ABB RAPID module: P80.mod

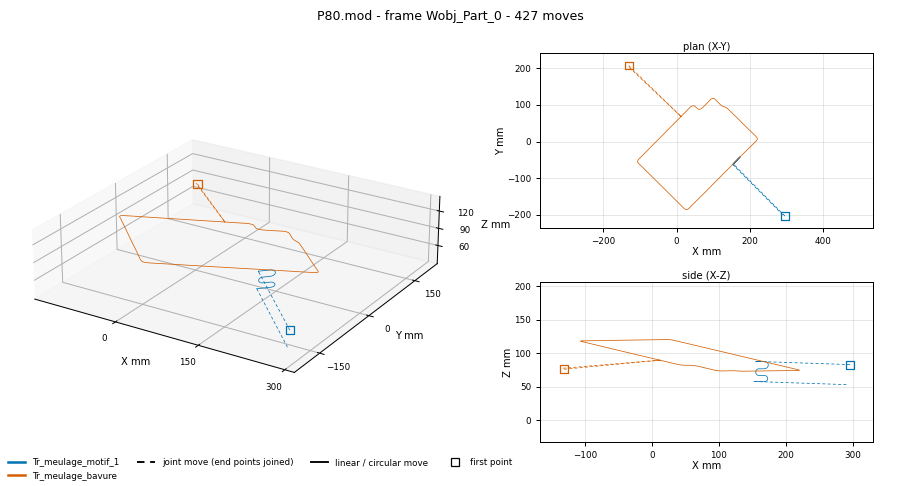
[picture p0: tool path of P80.mod in frame Wobj_Part_0, 427 of 434 moves have a stored position in this frame; points joined in program order, loops and branches not executed]
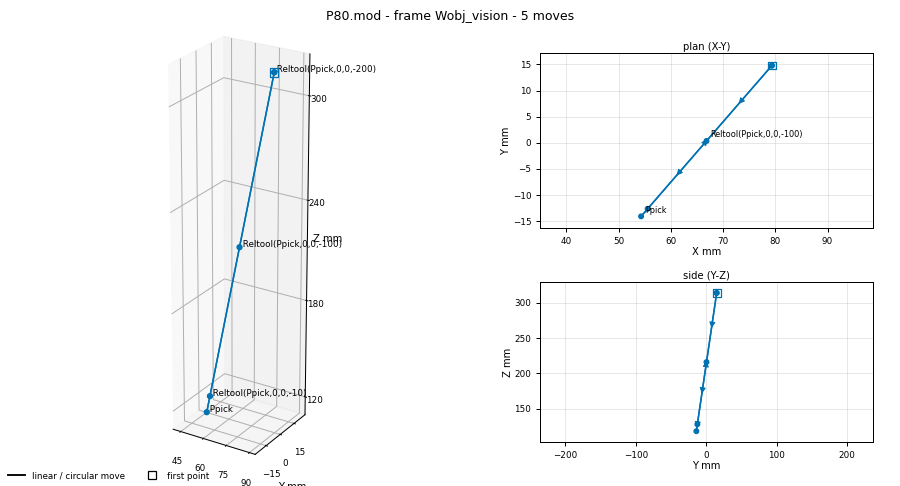
[picture p1: tool path of P80.mod in frame Wobj_vision, 5 of 434 moves have a stored position in this frame; points joined in program order, loops and branches not executed]
MODULE P80
	LOCAL CONST Speeddata vitesse_Tronconnage :=[10, 500, 0, 0];
	LOCAL CONST Robtarget Tr_meulage_motif_1_App1 :=[[295.968307149887,-203.258531598382,82.8714237887279],[0.661524902437711,-0.645987349747704,-0.266117883007714,0.272518659478957],[0,0,0,0],[8.999999E+09,8.999999E+09,8.999999E+09,8.999999E+09,8.999999E+09,8.999999E+09]];
	LOCAL CONST Robtarget Tr_meulage_motif_1_App2 :=[[162.175166138744,-68.4289722830441,87.3864379863114],[0.661524902437711,-0.645987349747704,-0.266117883007714,0.272518659478957],[0,0,0,0],[8.999999E+09,8.999999E+09,8.999999E+09,8.999999E+09,8.999999E+09,8.999999E+09]];
	LOCAL CONST Robtarget Tr_meulage_motif_1_P0 :=[[155.133421875,-61.3326796875,87.6240703125],[0.661524902437711,-0.645987349747704,-0.266117883007714,0.272518659478957],[0,0,0,0],[8.999999E+09,8.999999E+09,8.999999E+09,8.999999E+09,8.999999E+09,8.999999E+09]];
	LOCAL CONST Robtarget Tr_meulage_motif_1_P1 :=[[155.832390625,-60.61752734375,87.6240546875],[0.661524902437711,-0.645987349747704,-0.266117883007714,0.272518659478957],[0,0,0,0],[8.999999E+09,8.999999E+09,8.999999E+09,8.999999E+09,8.999999E+09,8.999999E+09]];
	LOCAL CONST Robtarget Tr_meulage_motif_1_P2 :=[[156.531359375,-59.902375,87.6240390625],[0.661524902437711,-0.645987349747704,-0.266117883007714,0.272518659478957],[0,0,0,0],[8.999999E+09,8.999999E+09,8.999999E+09,8.999999E+09,8.999999E+09,8.999999E+09]];
	LOCAL CONST Robtarget Tr_meulage_motif_1_P3 :=[[157.230328125,-59.18722265625,87.6240234375],[0.661524902437711,-0.645987349747704,-0.266117883007714,0.272518659478957],[0,0,0,0],[8.999999E+09,8.999999E+09,8.999999E+09,8.999999E+09,8.999999E+09,8.999999E+09]];
	LOCAL CONST Robtarget Tr_meulage_motif_1_P4 :=[[157.929296875,-58.47207421875,87.6240078125],[0.661524902437711,-0.645987349747704,-0.266117883007714,0.272518659478957],[0,0,0,0],[8.999999E+09,8.999999E+09,8.999999E+09,8.999999E+09,8.999999E+09,8.999999E+09]];
	LOCAL CONST Robtarget Tr_meulage_motif_1_P5 :=[[158.628265625,-57.756921875,87.6239921875],[0.661524902437711,-0.645987349747704,-0.266117883007714,0.272518659478957],[0,0,0,0],[8.999999E+09,8.999999E+09,8.999999E+09,8.999999E+09,8.999999E+09,8.999999E+09]];
	LOCAL CONST Robtarget Tr_meulage_motif_1_P6 :=[[159.327234375,-57.04176953125,87.6239765625],[0.661524902437711,-0.645987349747704,-0.266117883007714,0.272518659478957],[0,0,0,0],[8.999999E+09,8.999999E+09,8.999999E+09,8.999999E+09,8.999999E+09,8.999999E+09]];
	LOCAL CONST Robtarget Tr_meulage_motif_1_P7 :=[[160.026203125,-56.3266171875,87.6239609375],[0.661524902437711,-0.645987349747704,-0.266117883007714,0.272518659478957],[0,0,0,0],[8.999999E+09,8.999999E+09,8.999999E+09,8.999999E+09,8.999999E+09,8.999999E+09]];
	LOCAL CONST Robtarget Tr_meulage_motif_1_P8 :=[[160.725171875,-55.61146484375,87.6239453125],[0.661524902437711,-0.645987349747704,-0.266117883007714,0.272518659478957],[0,0,0,0],[8.999999E+09,8.999999E+09,8.999999E+09,8.999999E+09,8.999999E+09,8.999999E+09]];
	LOCAL CONST Robtarget Tr_meulage_motif_1_P9 :=[[161.424140625,-54.8963125,87.6239296875],[0.661524902437711,-0.645987349747704,-0.266117883007714,0.272518659478957],[0,0,0,0],[8.999999E+09,8.999999E+09,8.999999E+09,8.999999E+09,8.999999E+09,8.999999E+09]];
	LOCAL CONST Robtarget Tr_meulage_motif_1_P10 :=[[162.123109375,-54.1811640625,87.6239140625],[0.661524902437711,-0.645987349747704,-0.266117883007714,0.272518659478957],[0,0,0,0],[8.999999E+09,8.999999E+09,8.999999E+09,8.999999E+09,8.999999E+09,8.999999E+09]];
	LOCAL CONST Robtarget Tr_meulage_motif_1_P11 :=[[162.822078125,-53.46601171875,87.623890625],[0.661524902437711,-0.645987349747704,-0.266117883007714,0.272518659478957],[0,0,0,0],[8.999999E+09,8.999999E+09,8.999999E+09,8.999999E+09,8.999999E+09,8.999999E+09]];
	LOCAL CONST Robtarget Tr_meulage_motif_1_P12 :=[[163.521046875,-52.750859375,87.623875],[0.661524902437711,-0.645987349747704,-0.266117883007714,0.272518659478957],[0,0,0,0],[8.999999E+09,8.999999E+09,8.999999E+09,8.999999E+09,8.999999E+09,8.999999E+09]];
	LOCAL CONST Robtarget Tr_meulage_motif_1_P13 :=[[164.220015625,-52.03570703125,87.623859375],[0.661524902437711,-0.645987349747704,-0.266117883007714,0.272518659478957],[0,0,0,0],[8.999999E+09,8.999999E+09,8.999999E+09,8.999999E+09,8.999999E+09,8.999999E+09]];
	LOCAL CONST Robtarget Tr_meulage_motif_1_P14 :=[[164.918984375,-51.3205546875,87.62384375],[0.661524902437711,-0.645987349747704,-0.266117883007714,0.272518659478957],[0,0,0,0],[8.999999E+09,8.999999E+09,8.999999E+09,8.999999E+09,8.999999E+09,8.999999E+09]];
	LOCAL CONST Robtarget Tr_meulage_motif_1_P15 :=[[165.617953125,-50.60540625,87.623828125],[0.661524902437711,-0.645987349747704,-0.266117883007714,0.272518659478957],[0,0,0,0],[8.999999E+09,8.999999E+09,8.999999E+09,8.999999E+09,8.999999E+09,8.999999E+09]];
	LOCAL CONST Robtarget Tr_meulage_motif_1_P16 :=[[166.316921875,-49.89025390625,87.6238125],[0.661524902437711,-0.645987349747704,-0.266117883007714,0.272518659478957],[0,0,0,0],[8.999999E+09,8.999999E+09,8.999999E+09,8.999999E+09,8.999999E+09,8.999999E+09]];
	LOCAL CONST Robtarget Tr_meulage_motif_1_P17 :=[[167.015890625,-49.1751015625,87.623796875],[0.661524902437711,-0.645987349747704,-0.266117883007714,0.272518659478957],[0,0,0,0],[8.999999E+09,8.999999E+09,8.999999E+09,8.999999E+09,8.999999E+09,8.999999E+09]];
	LOCAL CONST Robtarget Tr_meulage_motif_1_P18 :=[[167.714859375,-48.45994921875,87.62378125],[0.661524902437711,-0.645987349747704,-0.266117883007714,0.272518659478957],[0,0,0,0],[8.999999E+09,8.999999E+09,8.999999E+09,8.999999E+09,8.999999E+09,8.999999E+09]];
	LOCAL CONST Robtarget Tr_meulage_motif_1_P19 :=[[168.413828125,-47.744796875,87.623765625],[0.661524902437711,-0.645987349747704,-0.266117883007714,0.272518659478957],[0,0,0,0],[8.999999E+09,8.999999E+09,8.999999E+09,8.999999E+09,8.999999E+09,8.999999E+09]];
	LOCAL CONST Robtarget Tr_meulage_motif_1_P20 :=[[169.1128125,-47.0296484375,87.62375],[0.661524902437711,-0.645987349747704,-0.266117883007714,0.272518659478957],[0,0,0,0],[8.999999E+09,8.999999E+09,8.999999E+09,8.999999E+09,8.999999E+09,8.999999E+09]];
	LOCAL CONST Robtarget Tr_meulage_motif_1_P21 :=[[169.80340625,-46.31671484375,87.5132265625],[0.661524902437711,-0.645987349747704,-0.266117883007714,0.272518659478957],[0,0,0,0],[8.999999E+09,8.999999E+09,8.999999E+09,8.999999E+09,8.999999E+09,8.999999E+09]];
	LOCAL CONST Robtarget Tr_meulage_motif_1_P22 :=[[170.458921875,-45.63391015625,87.3021953125],[0.661524902437711,-0.645987349747704,-0.266117883007714,0.272518659478957],[0,0,0,0],[8.999999E+09,8.999999E+09,8.999999E+09,8.999999E+09,8.999999E+09,8.999999E+09]];
	LOCAL CONST Robtarget Tr_meulage_motif_1_P23 :=[[171.047140625,-45.01647265625,87.0305546875],[0.661524902437711,-0.645987349747704,-0.266117883007714,0.272518659478957],[0,0,0,0],[8.999999E+09,8.999999E+09,8.999999E+09,8.999999E+09,8.999999E+09,8.999999E+09]];
	LOCAL CONST Robtarget Tr_meulage_motif_1_P24 :=[[171.563421875,-44.47242578125,86.754828125],[0.661524902437711,-0.645987349747704,-0.266117883007714,0.272518659478957],[0,0,0,0],[8.999999E+09,8.999999E+09,8.999999E+09,8.999999E+09,8.999999E+09,8.999999E+09]];
	LOCAL CONST Robtarget Tr_meulage_motif_1_P25 :=[[172.315359375,-43.66773828125,86.1391796875],[0.661524902437711,-0.645987349747704,-0.266117883007714,0.272518659478957],[0,0,0,0],[8.999999E+09,8.999999E+09,8.999999E+09,8.999999E+09,8.999999E+09,8.999999E+09]];
	LOCAL CONST Robtarget Tr_meulage_motif_1_P26 :=[[173.006703125,-42.91176953125,85.2921953125],[0.661524902437711,-0.645987349747704,-0.266117883007714,0.272518659478957],[0,0,0,0],[8.999999E+09,8.999999E+09,8.999999E+09,8.999999E+09,8.999999E+09,8.999999E+09]];
	LOCAL CONST Robtarget Tr_meulage_motif_1_P27 :=[[173.5698125,-42.27688671875,84.269125],[0.661524902437711,-0.645987349747704,-0.266117883007714,0.272518659478957],[0,0,0,0],[8.999999E+09,8.999999E+09,8.999999E+09,8.999999E+09,8.999999E+09,8.999999E+09]];
	LOCAL CONST Robtarget Tr_meulage_motif_1_P28 :=[[173.879015625,-41.896515625,83.153828125],[0.661524902437711,-0.645987349747704,-0.266117883007714,0.272518659478957],[0,0,0,0],[8.999999E+09,8.999999E+09,8.999999E+09,8.999999E+09,8.999999E+09,8.999999E+09]];
	LOCAL CONST Robtarget Tr_meulage_motif_1_P29 :=[[173.87796875,-41.85766796875,82.458421875],[0.661524902437711,-0.645987349747704,-0.266117883007714,0.272518659478957],[0,0,0,0],[8.999999E+09,8.999999E+09,8.999999E+09,8.999999E+09,8.999999E+09,8.999999E+09]];
	LOCAL CONST Robtarget Tr_meulage_motif_1_P30 :=[[173.859,-41.83914453125,81.797703125],[0.661524902437711,-0.645987349747704,-0.266117883007714,0.272518659478957],[0,0,0,0],[8.999999E+09,8.999999E+09,8.999999E+09,8.999999E+09,8.999999E+09,8.999999E+09]];
	LOCAL CONST Robtarget Tr_meulage_motif_1_P31 :=[[173.801671875,-41.85987109375,81.137140625],[0.661524902437711,-0.645987349747704,-0.266117883007714,0.272518659478957],[0,0,0,0],[8.999999E+09,8.999999E+09,8.999999E+09,8.999999E+09,8.999999E+09,8.999999E+09]];
	LOCAL CONST Robtarget Tr_meulage_motif_1_P32 :=[[173.42184375,-42.1853125,80.03628125],[0.661524902437711,-0.645987349747704,-0.266117883007714,0.272518659478957],[0,0,0,0],[8.999999E+09,8.999999E+09,8.999999E+09,8.999999E+09,8.999999E+09,8.999999E+09]];
	LOCAL CONST Robtarget Tr_meulage_motif_1_P33 :=[[172.79421875,-42.76973046875,79.030484375],[0.661524902437711,-0.645987349747704,-0.266117883007714,0.272518659478957],[0,0,0,0],[8.999999E+09,8.999999E+09,8.999999E+09,8.999999E+09,8.999999E+09,8.999999E+09]];
	LOCAL CONST Robtarget Tr_meulage_motif_1_P34 :=[[172.055109375,-43.47840625,78.2022890625],[0.661524902437711,-0.645987349747704,-0.266117883007714,0.272518659478957],[0,0,0,0],[8.999999E+09,8.999999E+09,8.999999E+09,8.999999E+09,8.999999E+09,8.999999E+09]];
	LOCAL CONST Robtarget Tr_meulage_motif_1_P35 :=[[171.5635,-43.9586953125,77.8068671875],[0.661524902437711,-0.645987349747704,-0.266117883007714,0.272518659478957],[0,0,0,0],[8.999999E+09,8.999999E+09,8.999999E+09,8.999999E+09,8.999999E+09,8.999999E+09]];
	LOCAL CONST Robtarget Tr_meulage_motif_1_P36 :=[[170.74,-44.773296875,77.31975],[0.661524902437711,-0.645987349747704,-0.266117883007714,0.272518659478957],[0,0,0,0],[8.999999E+09,8.999999E+09,8.999999E+09,8.999999E+09,8.999999E+09,8.999999E+09]];
	LOCAL CONST Robtarget Tr_meulage_motif_1_P37 :=[[170.14178125,-45.3702265625,77.0558828125],[0.661524902437711,-0.645987349747704,-0.266117883007714,0.272518659478957],[0,0,0,0],[8.999999E+09,8.999999E+09,8.999999E+09,8.999999E+09,8.999999E+09,8.999999E+09]];
	LOCAL CONST Robtarget Tr_meulage_motif_1_P38 :=[[169.48446875,-46.03101953125,76.85159375],[0.661524902437711,-0.645987349747704,-0.266117883007714,0.272518659478957],[0,0,0,0],[8.999999E+09,8.999999E+09,8.999999E+09,8.999999E+09,8.999999E+09,8.999999E+09]];
	LOCAL CONST Robtarget Tr_meulage_motif_1_P39 :=[[168.795265625,-46.72994140625,76.7431015625],[0.661524902437711,-0.645987349747704,-0.266117883007714,0.272518659478957],[0,0,0,0],[8.999999E+09,8.999999E+09,8.999999E+09,8.999999E+09,8.999999E+09,8.999999E+09]];
	LOCAL CONST Robtarget Tr_meulage_motif_1_P40 :=[[168.098328125,-47.43667578125,76.632609375],[0.661524902437711,-0.645987349747704,-0.266117883007714,0.272518659478957],[0,0,0,0],[8.999999E+09,8.999999E+09,8.999999E+09,8.999999E+09,8.999999E+09,8.999999E+09]];
	LOCAL CONST Robtarget Tr_meulage_motif_1_P41 :=[[167.399359375,-48.151828125,76.632625],[0.661524902437711,-0.645987349747704,-0.266117883007714,0.272518659478957],[0,0,0,0],[8.999999E+09,8.999999E+09,8.999999E+09,8.999999E+09,8.999999E+09,8.999999E+09]];
	LOCAL CONST Robtarget Tr_meulage_motif_1_P42 :=[[166.700390625,-48.86698046875,76.632640625],[0.661524902437711,-0.645987349747704,-0.266117883007714,0.272518659478957],[0,0,0,0],[8.999999E+09,8.999999E+09,8.999999E+09,8.999999E+09,8.999999E+09,8.999999E+09]];
	LOCAL CONST Robtarget Tr_meulage_motif_1_P43 :=[[166.001421875,-49.5821328125,76.63265625],[0.661524902437711,-0.645987349747704,-0.266117883007714,0.272518659478957],[0,0,0,0],[8.999999E+09,8.999999E+09,8.999999E+09,8.999999E+09,8.999999E+09,8.999999E+09]];
	LOCAL CONST Robtarget Tr_meulage_motif_1_P44 :=[[165.302453125,-50.29728515625,76.632671875],[0.661524902437711,-0.645987349747704,-0.266117883007714,0.272518659478957],[0,0,0,0],[8.999999E+09,8.999999E+09,8.999999E+09,8.999999E+09,8.999999E+09,8.999999E+09]];
	LOCAL CONST Robtarget Tr_meulage_motif_1_P45 :=[[164.603484375,-51.01243359375,76.6326875],[0.661524902437711,-0.645987349747704,-0.266117883007714,0.272518659478957],[0,0,0,0],[8.999999E+09,8.999999E+09,8.999999E+09,8.999999E+09,8.999999E+09,8.999999E+09]];
	LOCAL CONST Robtarget Tr_meulage_motif_1_P46 :=[[163.904515625,-51.7275859375,76.632703125],[0.661524902437711,-0.645987349747704,-0.266117883007714,0.272518659478957],[0,0,0,0],[8.999999E+09,8.999999E+09,8.999999E+09,8.999999E+09,8.999999E+09,8.999999E+09]];
	LOCAL CONST Robtarget Tr_meulage_motif_1_P47 :=[[163.205546875,-52.44273828125,76.63271875],[0.661524902437711,-0.645987349747704,-0.266117883007714,0.272518659478957],[0,0,0,0],[8.999999E+09,8.999999E+09,8.999999E+09,8.999999E+09,8.999999E+09,8.999999E+09]];
	LOCAL CONST Robtarget Tr_meulage_motif_1_P48 :=[[162.506578125,-53.157890625,76.632734375],[0.661524902437711,-0.645987349747704,-0.266117883007714,0.272518659478957],[0,0,0,0],[8.999999E+09,8.999999E+09,8.999999E+09,8.999999E+09,8.999999E+09,8.999999E+09]];
	LOCAL CONST Robtarget Tr_meulage_motif_1_P49 :=[[161.807609375,-53.87304296875,76.6327578125],[0.661524902437711,-0.645987349747704,-0.266117883007714,0.272518659478957],[0,0,0,0],[8.999999E+09,8.999999E+09,8.999999E+09,8.999999E+09,8.999999E+09,8.999999E+09]];
	LOCAL CONST Robtarget Tr_meulage_motif_1_P50 :=[[161.108640625,-54.58819140625,76.6327734375],[0.661524902437711,-0.645987349747704,-0.266117883007714,0.272518659478957],[0,0,0,0],[8.999999E+09,8.999999E+09,8.999999E+09,8.999999E+09,8.999999E+09,8.999999E+09]];
	LOCAL CONST Robtarget Tr_meulage_motif_1_P51 :=[[160.409671875,-55.30334375,76.6327890625],[0.661524902437711,-0.645987349747704,-0.266117883007714,0.272518659478957],[0,0,0,0],[8.999999E+09,8.999999E+09,8.999999E+09,8.999999E+09,8.999999E+09,8.999999E+09]];
	LOCAL CONST Robtarget Tr_meulage_motif_1_P52 :=[[159.710703125,-56.01849609375,76.6328046875],[0.661524902437711,-0.645987349747704,-0.266117883007714,0.272518659478957],[0,0,0,0],[8.999999E+09,8.999999E+09,8.999999E+09,8.999999E+09,8.999999E+09,8.999999E+09]];
	LOCAL CONST Robtarget Tr_meulage_motif_1_P53 :=[[159.01375,-56.72523046875,76.5223125],[0.661524902437711,-0.645987349747704,-0.266117883007714,0.272518659478957],[0,0,0,0],[8.999999E+09,8.999999E+09,8.999999E+09,8.999999E+09,8.999999E+09,8.999999E+09]];
	LOCAL CONST Robtarget Tr_meulage_motif_1_P54 :=[[158.346125,-57.39620703125,76.3113125],[0.661524902437711,-0.645987349747704,-0.266117883007714,0.272518659478957],[0,0,0,0],[8.999999E+09,8.999999E+09,8.999999E+09,8.999999E+09,8.999999E+09,8.999999E+09]];
	LOCAL CONST Robtarget Tr_meulage_motif_1_P55 :=[[157.742296875,-57.9984140625,76.0396953125],[0.661524902437711,-0.645987349747704,-0.266117883007714,0.272518659478957],[0,0,0,0],[8.999999E+09,8.999999E+09,8.999999E+09,8.999999E+09,8.999999E+09,8.999999E+09]];
	LOCAL CONST Robtarget Tr_meulage_motif_1_P56 :=[[157.236265625,-58.4987265625,75.735796875],[0.661524902437711,-0.645987349747704,-0.266117883007714,0.272518659478957],[0,0,0,0],[8.999999E+09,8.999999E+09,8.999999E+09,8.999999E+09,8.999999E+09,8.999999E+09]];
	LOCAL CONST Robtarget Tr_meulage_motif_1_P57 :=[[156.494203125,-59.21996875,75.0738125],[0.661524902437711,-0.645987349747704,-0.266117883007714,0.272518659478957],[0,0,0,0],[8.999999E+09,8.999999E+09,8.999999E+09,8.999999E+09,8.999999E+09,8.999999E+09]];
	LOCAL CONST Robtarget Tr_meulage_motif_1_P58 :=[[155.83790625,-59.8397265625,74.1726171875],[0.661524902437711,-0.645987349747704,-0.266117883007714,0.272518659478957],[0,0,0,0],[8.999999E+09,8.999999E+09,8.999999E+09,8.999999E+09,8.999999E+09,8.999999E+09]];
	LOCAL CONST Robtarget Tr_meulage_motif_1_P59 :=[[155.43396875,-60.19301171875,73.1274375],[0.661524902437711,-0.645987349747704,-0.266117883007714,0.272518659478957],[0,0,0,0],[8.999999E+09,8.999999E+09,8.999999E+09,8.999999E+09,8.999999E+09,8.999999E+09]];
	LOCAL CONST Robtarget Tr_meulage_motif_1_P60 :=[[155.2849375,-60.30573828125,72.43478125],[0.661524902437711,-0.645987349747704,-0.266117883007714,0.272518659478957],[0,0,0,0],[8.999999E+09,8.999999E+09,8.999999E+09,8.999999E+09,8.999999E+09,8.999999E+09]];
	LOCAL CONST Robtarget Tr_meulage_motif_1_P61 :=[[155.21821875,-60.329828125,71.6653984375],[0.661524902437711,-0.645987349747704,-0.266117883007714,0.272518659478957],[0,0,0,0],[8.999999E+09,8.999999E+09,8.999999E+09,8.999999E+09,8.999999E+09,8.999999E+09]];
	LOCAL CONST Robtarget Tr_meulage_motif_1_P62 :=[[155.242921875,-60.26039453125,70.896140625],[0.661524902437711,-0.645987349747704,-0.266117883007714,0.272518659478957],[0,0,0,0],[8.999999E+09,8.999999E+09,8.999999E+09,8.999999E+09,8.999999E+09,8.999999E+09]];
	LOCAL CONST Robtarget Tr_meulage_motif_1_P63 :=[[155.504421875,-59.92927734375,69.7887734375],[0.661524902437711,-0.645987349747704,-0.266117883007714,0.272518659478957],[0,0,0,0],[8.999999E+09,8.999999E+09,8.999999E+09,8.999999E+09,8.999999E+09,8.999999E+09]];
	LOCAL CONST Robtarget Tr_meulage_motif_1_P64 :=[[155.77721875,-59.61657421875,69.2035546875],[0.661524902437711,-0.645987349747704,-0.266117883007714,0.272518659478957],[0,0,0,0],[8.999999E+09,8.999999E+09,8.999999E+09,8.999999E+09,8.999999E+09,8.999999E+09]];
	LOCAL CONST Robtarget Tr_meulage_motif_1_P65 :=[[156.37184375,-58.957296875,68.317125],[0.661524902437711,-0.645987349747704,-0.266117883007714,0.272518659478957],[0,0,0,0],[8.999999E+09,8.999999E+09,8.999999E+09,8.999999E+09,8.999999E+09,8.999999E+09]];
	LOCAL CONST Robtarget Tr_meulage_motif_1_P66 :=[[156.76934375,-58.5268359375,67.903140625],[0.661524902437711,-0.645987349747704,-0.266117883007714,0.272518659478957],[0,0,0,0],[8.999999E+09,8.999999E+09,8.999999E+09,8.999999E+09,8.999999E+09,8.999999E+09]];
	LOCAL CONST Robtarget Tr_meulage_motif_1_P67 :=[[157.535109375,-57.712125,67.3594609375],[0.661524902437711,-0.645987349747704,-0.266117883007714,0.272518659478957],[0,0,0,0],[8.999999E+09,8.999999E+09,8.999999E+09,8.999999E+09,8.999999E+09,8.999999E+09]];
	LOCAL CONST Robtarget Tr_meulage_motif_1_P68 :=[[158.103703125,-57.113421875,67.0641875],[0.661524902437711,-0.645987349747704,-0.266117883007714,0.272518659478957],[0,0,0,0],[8.999999E+09,8.999999E+09,8.999999E+09,8.999999E+09,8.999999E+09,8.999999E+09]];
	LOCAL CONST Robtarget Tr_meulage_motif_1_P69 :=[[158.74928125,-56.441171875,66.8598671875],[0.661524902437711,-0.645987349747704,-0.266117883007714,0.272518659478957],[0,0,0,0],[8.999999E+09,8.999999E+09,8.999999E+09,8.999999E+09,8.999999E+09,8.999999E+09]];
	LOCAL CONST Robtarget Tr_meulage_motif_1_P70 :=[[159.43225,-55.7361640625,66.75134375],[0.661524902437711,-0.645987349747704,-0.266117883007714,0.272518659478957],[0,0,0,0],[8.999999E+09,8.999999E+09,8.999999E+09,8.999999E+09,8.999999E+09,8.999999E+09]];
	LOCAL CONST Robtarget Tr_meulage_motif_1_P71 :=[[160.12284375,-55.023234375,66.640828125],[0.661524902437711,-0.645987349747704,-0.266117883007714,0.272518659478957],[0,0,0,0],[8.999999E+09,8.999999E+09,8.999999E+09,8.999999E+09,8.999999E+09,8.999999E+09]];
	LOCAL CONST Robtarget Tr_meulage_motif_1_P72 :=[[160.8218125,-54.30808203125,66.6408125],[0.661524902437711,-0.645987349747704,-0.266117883007714,0.272518659478957],[0,0,0,0],[8.999999E+09,8.999999E+09,8.999999E+09,8.999999E+09,8.999999E+09,8.999999E+09]];
	LOCAL CONST Robtarget Tr_meulage_motif_1_P73 :=[[161.52078125,-53.59293359375,66.640796875],[0.661524902437711,-0.645987349747704,-0.266117883007714,0.272518659478957],[0,0,0,0],[8.999999E+09,8.999999E+09,8.999999E+09,8.999999E+09,8.999999E+09,8.999999E+09]];
	LOCAL CONST Robtarget Tr_meulage_motif_1_P74 :=[[162.21975,-52.87778125,66.64078125],[0.661524902437711,-0.645987349747704,-0.266117883007714,0.272518659478957],[0,0,0,0],[8.999999E+09,8.999999E+09,8.999999E+09,8.999999E+09,8.999999E+09,8.999999E+09]];
	LOCAL CONST Robtarget Tr_meulage_motif_1_P75 :=[[162.91871875,-52.16262890625,66.640765625],[0.661524902437711,-0.645987349747704,-0.266117883007714,0.272518659478957],[0,0,0,0],[8.999999E+09,8.999999E+09,8.999999E+09,8.999999E+09,8.999999E+09,8.999999E+09]];
	LOCAL CONST Robtarget Tr_meulage_motif_1_P76 :=[[163.6176875,-51.4474765625,66.6407421875],[0.661524902437711,-0.645987349747704,-0.266117883007714,0.272518659478957],[0,0,0,0],[8.999999E+09,8.999999E+09,8.999999E+09,8.999999E+09,8.999999E+09,8.999999E+09]];
	LOCAL CONST Robtarget Tr_meulage_motif_1_P77 :=[[164.31665625,-50.73232421875,66.6407265625],[0.661524902437711,-0.645987349747704,-0.266117883007714,0.272518659478957],[0,0,0,0],[8.999999E+09,8.999999E+09,8.999999E+09,8.999999E+09,8.999999E+09,8.999999E+09]];
	LOCAL CONST Robtarget Tr_meulage_motif_1_P78 :=[[165.015625,-50.01717578125,66.6407109375],[0.661524902437711,-0.645987349747704,-0.266117883007714,0.272518659478957],[0,0,0,0],[8.999999E+09,8.999999E+09,8.999999E+09,8.999999E+09,8.999999E+09,8.999999E+09]];
	LOCAL CONST Robtarget Tr_meulage_motif_1_P79 :=[[165.71459375,-49.3020234375,66.6406953125],[0.661524902437711,-0.645987349747704,-0.266117883007714,0.272518659478957],[0,0,0,0],[8.999999E+09,8.999999E+09,8.999999E+09,8.999999E+09,8.999999E+09,8.999999E+09]];
	LOCAL CONST Robtarget Tr_meulage_motif_1_P80 :=[[166.4135625,-48.58687109375,66.6406796875],[0.661524902437711,-0.645987349747704,-0.266117883007714,0.272518659478957],[0,0,0,0],[8.999999E+09,8.999999E+09,8.999999E+09,8.999999E+09,8.999999E+09,8.999999E+09]];
	LOCAL CONST Robtarget Tr_meulage_motif_1_P81 :=[[167.11253125,-47.87171875,66.6406640625],[0.661524902437711,-0.645987349747704,-0.266117883007714,0.272518659478957],[0,0,0,0],[8.999999E+09,8.999999E+09,8.999999E+09,8.999999E+09,8.999999E+09,8.999999E+09]];
	LOCAL CONST Robtarget Tr_meulage_motif_1_P82 :=[[167.8115,-47.15656640625,66.6406484375],[0.661524902437711,-0.645987349747704,-0.266117883007714,0.272518659478957],[0,0,0,0],[8.999999E+09,8.999999E+09,8.999999E+09,8.999999E+09,8.999999E+09,8.999999E+09]];
	LOCAL CONST Robtarget Tr_meulage_motif_1_P83 :=[[168.51046875,-46.4414140625,66.6406328125],[0.661524902437711,-0.645987349747704,-0.266117883007714,0.272518659478957],[0,0,0,0],[8.999999E+09,8.999999E+09,8.999999E+09,8.999999E+09,8.999999E+09,8.999999E+09]];
	LOCAL CONST Robtarget Tr_meulage_motif_1_P84 :=[[169.201078125,-45.728484375,66.530109375],[0.661524902437711,-0.645987349747704,-0.266117883007714,0.272518659478957],[0,0,0,0],[8.999999E+09,8.999999E+09,8.999999E+09,8.999999E+09,8.999999E+09,8.999999E+09]];
	LOCAL CONST Robtarget Tr_meulage_motif_1_P85 :=[[169.85659375,-45.0456796875,66.319078125],[0.661524902437711,-0.645987349747704,-0.266117883007714,0.272518659478957],[0,0,0,0],[8.999999E+09,8.999999E+09,8.999999E+09,8.999999E+09,8.999999E+09,8.999999E+09]];
	LOCAL CONST Robtarget Tr_meulage_motif_1_P86 :=[[170.4448125,-44.4282421875,66.0474453125],[0.661524902437711,-0.645987349747704,-0.266117883007714,0.272518659478957],[0,0,0,0],[8.999999E+09,8.999999E+09,8.999999E+09,8.999999E+09,8.999999E+09,8.999999E+09]];
	LOCAL CONST Robtarget Tr_meulage_motif_1_P87 :=[[170.96109375,-43.88419140625,65.7717109375],[0.661524902437711,-0.645987349747704,-0.266117883007714,0.272518659478957],[0,0,0,0],[8.999999E+09,8.999999E+09,8.999999E+09,8.999999E+09,8.999999E+09,8.999999E+09]];
	LOCAL CONST Robtarget Tr_meulage_motif_1_P88 :=[[171.71303125,-43.0795078125,65.15606640625],[0.661524902437711,-0.645987349747704,-0.266117883007714,0.272518659478957],[0,0,0,0],[8.999999E+09,8.999999E+09,8.999999E+09,8.999999E+09,8.999999E+09,8.999999E+09]];
	LOCAL CONST Robtarget Tr_meulage_motif_1_P89 :=[[172.404375,-42.3235390625,64.30907421875],[0.661524902437711,-0.645987349747704,-0.266117883007714,0.272518659478957],[0,0,0,0],[8.999999E+09,8.999999E+09,8.999999E+09,8.999999E+09,8.999999E+09,8.999999E+09]];
	LOCAL CONST Robtarget Tr_meulage_motif_1_P90 :=[[172.89975,-41.7556015625,63.24498046875],[0.661524902437711,-0.645987349747704,-0.266117883007714,0.272518659478957],[0,0,0,0],[8.999999E+09,8.999999E+09,8.999999E+09,8.999999E+09,8.999999E+09,8.999999E+09]];
	LOCAL CONST Robtarget Tr_meulage_motif_1_P91 :=[[173.087890625,-41.50144140625,62.17071484375],[0.661524902437711,-0.645987349747704,-0.266117883007714,0.272518659478957],[0,0,0,0],[8.999999E+09,8.999999E+09,8.999999E+09,8.999999E+09,8.999999E+09,8.999999E+09]];
	LOCAL CONST Robtarget Tr_meulage_motif_1_P92 :=[[173.030015625,-41.5273515625,61.59058984375],[0.661524902437711,-0.645987349747704,-0.266117883007714,0.272518659478957],[0,0,0,0],[8.999999E+09,8.999999E+09,8.999999E+09,8.999999E+09,8.999999E+09,8.999999E+09]];
	LOCAL CONST Robtarget Tr_meulage_motif_1_P93 :=[[173.021046875,-41.5125625,61.17301953125],[0.661524902437711,-0.645987349747704,-0.266117883007714,0.272518659478957],[0,0,0,0],[8.999999E+09,8.999999E+09,8.999999E+09,8.999999E+09,8.999999E+09,8.999999E+09]];
	LOCAL CONST Robtarget Tr_meulage_motif_1_P94 :=[[172.740109375,-41.74440625,60.2044921875],[0.661524902437711,-0.645987349747704,-0.266117883007714,0.272518659478957],[0,0,0,0],[8.999999E+09,8.999999E+09,8.999999E+09,8.999999E+09,8.999999E+09,8.999999E+09]];
	LOCAL CONST Robtarget Tr_meulage_motif_1_P95 :=[[172.13928125,-42.30651171875,59.2875859375],[0.661524902437711,-0.645987349747704,-0.266117883007714,0.272518659478957],[0,0,0,0],[8.999999E+09,8.999999E+09,8.999999E+09,8.999999E+09,8.999999E+09,8.999999E+09]];
	LOCAL CONST Robtarget Tr_meulage_motif_1_P96 :=[[171.699265625,-42.73244921875,58.865],[0.661524902437711,-0.645987349747704,-0.266117883007714,0.272518659478957],[0,0,0,0],[8.999999E+09,8.999999E+09,8.999999E+09,8.999999E+09,8.999999E+09,8.999999E+09]];
	LOCAL CONST Robtarget Tr_meulage_motif_1_P97 :=[[170.894,-43.5259375,58.3350078125],[0.661524902437711,-0.645987349747704,-0.266117883007714,0.272518659478957],[0,0,0,0],[8.999999E+09,8.999999E+09,8.999999E+09,8.999999E+09,8.999999E+09,8.999999E+09]];
	LOCAL CONST Robtarget Tr_meulage_motif_1_P98 :=[[170.29578125,-44.12286328125,58.071140625],[0.661524902437711,-0.645987349747704,-0.266117883007714,0.272518659478957],[0,0,0,0],[8.999999E+09,8.999999E+09,8.999999E+09,8.999999E+09,8.999999E+09,8.999999E+09]];
	LOCAL CONST Robtarget Tr_meulage_motif_1_P99 :=[[169.63846875,-44.78365625,57.86684765625],[0.661524902437711,-0.645987349747704,-0.266117883007714,0.272518659478957],[0,0,0,0],[8.999999E+09,8.999999E+09,8.999999E+09,8.999999E+09,8.999999E+09,8.999999E+09]];
	LOCAL CONST Robtarget Tr_meulage_motif_1_P100 :=[[168.94928125,-45.48258203125,57.758359375],[0.661524902437711,-0.645987349747704,-0.266117883007714,0.272518659478957],[0,0,0,0],[8.999999E+09,8.999999E+09,8.999999E+09,8.999999E+09,8.999999E+09,8.999999E+09]];
	LOCAL CONST Robtarget Tr_meulage_motif_1_P101 :=[[168.252328125,-46.18931640625,57.64787109375],[0.661524902437711,-0.645987349747704,-0.266117883007714,0.272518659478957],[0,0,0,0],[8.999999E+09,8.999999E+09,8.999999E+09,8.999999E+09,8.999999E+09,8.999999E+09]];
	LOCAL CONST Robtarget Tr_meulage_motif_1_P102 :=[[167.553359375,-46.90446875,57.64788671875],[0.661524902437711,-0.645987349747704,-0.266117883007714,0.272518659478957],[0,0,0,0],[8.999999E+09,8.999999E+09,8.999999E+09,8.999999E+09,8.999999E+09,8.999999E+09]];
	LOCAL CONST Robtarget Tr_meulage_motif_1_P103 :=[[166.854390625,-47.61962109375,57.64790234375],[0.661524902437711,-0.645987349747704,-0.266117883007714,0.272518659478957],[0,0,0,0],[8.999999E+09,8.999999E+09,8.999999E+09,8.999999E+09,8.999999E+09,8.999999E+09]];
	LOCAL CONST Robtarget Tr_meulage_motif_1_P104 :=[[166.155421875,-48.3347734375,57.64791796875],[0.661524902437711,-0.645987349747704,-0.266117883007714,0.272518659478957],[0,0,0,0],[8.999999E+09,8.999999E+09,8.999999E+09,8.999999E+09,8.999999E+09,8.999999E+09]];
	LOCAL CONST Robtarget Tr_meulage_motif_1_P105 :=[[165.456453125,-49.049921875,57.64793359375],[0.661524902437711,-0.645987349747704,-0.266117883007714,0.272518659478957],[0,0,0,0],[8.999999E+09,8.999999E+09,8.999999E+09,8.999999E+09,8.999999E+09,8.999999E+09]];
	LOCAL CONST Robtarget Tr_meulage_motif_1_P106 :=[[164.757484375,-49.76507421875,57.64794921875],[0.661524902437711,-0.645987349747704,-0.266117883007714,0.272518659478957],[0,0,0,0],[8.999999E+09,8.999999E+09,8.999999E+09,8.999999E+09,8.999999E+09,8.999999E+09]];
	LOCAL CONST Robtarget Tr_meulage_motif_1_P107 :=[[164.058515625,-50.4802265625,57.64796484375],[0.661524902437711,-0.645987349747704,-0.266117883007714,0.272518659478957],[0,0,0,0],[8.999999E+09,8.999999E+09,8.999999E+09,8.999999E+09,8.999999E+09,8.999999E+09]];
	LOCAL CONST Robtarget Tr_meulage_motif_1_P108 :=[[163.359546875,-51.19537890625,57.64798046875],[0.661524902437711,-0.645987349747704,-0.266117883007714,0.272518659478957],[0,0,0,0],[8.999999E+09,8.999999E+09,8.999999E+09,8.999999E+09,8.999999E+09,8.999999E+09]];
	LOCAL CONST Robtarget Tr_meulage_motif_1_P109 :=[[162.660578125,-51.91053125,57.64799609375],[0.661524902437711,-0.645987349747704,-0.266117883007714,0.272518659478957],[0,0,0,0],[8.999999E+09,8.999999E+09,8.999999E+09,8.999999E+09,8.999999E+09,8.999999E+09]];
	LOCAL CONST Robtarget Tr_meulage_motif_1_P110 :=[[161.961609375,-52.6256796875,57.64801171875],[0.661524902437711,-0.645987349747704,-0.266117883007714,0.272518659478957],[0,0,0,0],[8.999999E+09,8.999999E+09,8.999999E+09,8.999999E+09,8.999999E+09,8.999999E+09]];
	LOCAL CONST Robtarget Tr_meulage_motif_1_P111 :=[[161.262640625,-53.34083203125,57.64803125],[0.661524902437711,-0.645987349747704,-0.266117883007714,0.272518659478957],[0,0,0,0],[8.999999E+09,8.999999E+09,8.999999E+09,8.999999E+09,8.999999E+09,8.999999E+09]];
	LOCAL CONST Robtarget Tr_meulage_motif_1_P112 :=[[160.563671875,-54.055984375,57.648046875],[0.661524902437711,-0.645987349747704,-0.266117883007714,0.272518659478957],[0,0,0,0],[8.999999E+09,8.999999E+09,8.999999E+09,8.999999E+09,8.999999E+09,8.999999E+09]];
	LOCAL CONST Robtarget Tr_meulage_motif_1_P113 :=[[159.864703125,-54.77113671875,57.6480625],[0.661524902437711,-0.645987349747704,-0.266117883007714,0.272518659478957],[0,0,0,0],[8.999999E+09,8.999999E+09,8.999999E+09,8.999999E+09,8.999999E+09,8.999999E+09]];
	LOCAL CONST Robtarget Tr_meulage_motif_1_P114 :=[[159.165734375,-55.4862890625,57.648078125],[0.661524902437711,-0.645987349747704,-0.266117883007714,0.272518659478957],[0,0,0,0],[8.999999E+09,8.999999E+09,8.999999E+09,8.999999E+09,8.999999E+09,8.999999E+09]];
	LOCAL CONST Robtarget Tr_meulage_motif_1_P115 :=[[158.466765625,-56.2014375,57.64809375],[0.661524902437711,-0.645987349747704,-0.266117883007714,0.272518659478957],[0,0,0,0],[8.999999E+09,8.999999E+09,8.999999E+09,8.999999E+09,8.999999E+09,8.999999E+09]];
	LOCAL CONST Robtarget Tr_meulage_motif_1_P116 :=[[157.767796875,-56.91658984375,57.648109375],[0.661524902437711,-0.645987349747704,-0.266117883007714,0.272518659478957],[0,0,0,0],[8.999999E+09,8.999999E+09,8.999999E+09,8.999999E+09,8.999999E+09,8.999999E+09]];
	LOCAL CONST Robtarget Tr_meulage_motif_1_P117 :=[[157.068828125,-57.6317421875,57.648125],[0.661524902437711,-0.645987349747704,-0.266117883007714,0.272518659478957],[0,0,0,0],[8.999999E+09,8.999999E+09,8.999999E+09,8.999999E+09,8.999999E+09,8.999999E+09]];
	LOCAL CONST Robtarget Tr_meulage_motif_1_P118 :=[[156.369859375,-58.34689453125,57.648140625],[0.661524902437711,-0.645987349747704,-0.266117883007714,0.272518659478957],[0,0,0,0],[8.999999E+09,8.999999E+09,8.999999E+09,8.999999E+09,8.999999E+09,8.999999E+09]];
	LOCAL CONST Robtarget Tr_meulage_motif_1_P119 :=[[155.670890625,-59.062046875,57.64815625],[0.661524902437711,-0.645987349747704,-0.266117883007714,0.272518659478957],[0,0,0,0],[8.999999E+09,8.999999E+09,8.999999E+09,8.999999E+09,8.999999E+09,8.999999E+09]];
	LOCAL CONST Robtarget Tr_meulage_motif_1_P120 :=[[154.971921875,-59.7771953125,57.648171875],[0.661524902437711,-0.645987349747704,-0.266117883007714,0.272518659478957],[0,0,0,0],[8.999999E+09,8.999999E+09,8.999999E+09,8.999999E+09,8.999999E+09,8.999999E+09]];
	LOCAL CONST Robtarget Tr_meulage_motif_1_P121 :=[[154.272953125,-60.49234765625,57.6481875],[0.661524902437711,-0.645987349747704,-0.266117883007714,0.272518659478957],[0,0,0,0],[8.999999E+09,8.999999E+09,8.999999E+09,8.999999E+09,8.999999E+09,8.999999E+09]];
	LOCAL CONST Robtarget Tr_meulage_motif_1_P122 :=[[153.573984375,-61.2075,57.64820703125],[0.661524902437711,-0.645987349747704,-0.266117883007714,0.272518659478957],[0,0,0,0],[8.999999E+09,8.999999E+09,8.999999E+09,8.999999E+09,8.999999E+09,8.999999E+09]];
	LOCAL CONST Robtarget Tr_meulage_motif_1_P123 :=[[152.875015625,-61.92265234375,57.64822265625],[0.661524902437711,-0.645987349747704,-0.266117883007714,0.272518659478957],[0,0,0,0],[8.999999E+09,8.999999E+09,8.999999E+09,8.999999E+09,8.999999E+09,8.999999E+09]];
	LOCAL CONST Robtarget Tr_meulage_motif_1_degg1 :=[[159.916759888744,-69.0189449392941,57.4105903300614],[0.661524902437711,-0.645987349747704,-0.266117883007714,0.272518659478957],[0,0,0,0],[8.999999E+09,8.999999E+09,8.999999E+09,8.999999E+09,8.999999E+09,8.999999E+09]];
	LOCAL CONST Robtarget Tr_meulage_motif_1_degg2 :=[[293.709900899887,-203.848504254632,52.8955761324779],[0.661524902437711,-0.645987349747704,-0.266117883007714,0.272518659478957],[0,0,0,0],[8.999999E+09,8.999999E+09,8.999999E+09,8.999999E+09,8.999999E+09,8.999999E+09]];
	LOCAL CONST Robtarget Tr_meulage_bavure_App1 :=[[-130.802481498914,207.516367832347,75.9567690677868],[0.284428212423492,-0.265826681388466,0.628943133613018,-0.672954160489858],[0,0,0,0],[8.999999E+09,8.999999E+09,8.999999E+09,8.999999E+09,8.999999E+09,8.999999E+09]];
	LOCAL CONST Robtarget Tr_meulage_bavure_App2 :=[[5.1532886203668,75.4126773759924,88.7881189221393],[0.284428212423492,-0.265826681388466,0.628943133613018,-0.672954160489858],[0,0,0,0],[8.999999E+09,8.999999E+09,8.999999E+09,8.999999E+09,8.999999E+09,8.999999E+09]];
	LOCAL CONST Robtarget Tr_meulage_bavure_P0 :=[[12.30885546875,68.4598515625,89.463453125],[0.284428212423492,-0.265826681388466,0.628943133613018,-0.672954160489858],[0,0,0,0],[8.999999E+09,8.999999E+09,8.999999E+09,8.999999E+09,8.999999E+09,8.999999E+09]];
	LOCAL CONST Robtarget Tr_meulage_bavure_P1 :=[[12.0715,68.21390625,89.5204921875],[0.284373042901133,-0.26576929181495,0.628958710011008,-0.672985584615762],[0,0,0,0],[8.999999E+09,8.999999E+09,8.999999E+09,8.999999E+09,8.999999E+09,8.999999E+09]];
	LOCAL CONST Robtarget Tr_meulage_bavure_P2 :=[[8.9287109375,65.15151953125,90.2510546875],[0.284222180764744,-0.265608224533555,0.62899684472372,-0.673077255854831],[0,0,0,0],[8.999999E+09,8.999999E+09,8.999999E+09,8.999999E+09,8.999999E+09,8.999999E+09]];
	LOCAL CONST Robtarget Tr_meulage_bavure_P3 :=[[4.699265625,60.7726875,91.266953125],[0.284001346399506,-0.26537480227308,0.629055039986907,-0.673208144802825],[0,0,0,0],[8.999999E+09,8.999999E+09,8.999999E+09,8.999999E+09,8.999999E+09,8.999999E+09]];
	LOCAL CONST Robtarget Tr_meulage_bavure_P4 :=[[3.99077392578125,60.0665703125,91.4336484375],[0.283733376273213,-0.265091369093486,0.629125242398549,-0.673367185566472],[0,0,0,0],[8.999999E+09,8.999999E+09,8.999999E+09,8.999999E+09,8.999999E+09,8.999999E+09]];
	LOCAL CONST Robtarget Tr_meulage_bavure_P5 :=[[3.88059838867188,59.94528125,91.46103125],[0.28347686519291,-0.264814256821455,0.629186003163786,-0.673527467670979],[0,0,0,0],[8.999999E+09,8.999999E+09,8.999999E+09,8.999999E+09,8.999999E+09,8.999999E+09]];
	LOCAL CONST Robtarget Tr_meulage_bavure_P6 :=[[3.76301000976563,59.827015625,91.488828125],[0.283331719588849,-0.264646166761516,0.629208160231015,-0.673633902199083],[0,0,0,0],[8.999999E+09,8.999999E+09,8.999999E+09,8.999999E+09,8.999999E+09,8.999999E+09]];
	LOCAL CONST Robtarget Tr_meulage_bavure_P7 :=[[3.63213793945313,59.70169921875,91.51896875],[0.283479615359356,-0.264761899820276,0.629125995315525,-0.673602943949564],[0,0,0,0],[8.999999E+09,8.999999E+09,8.999999E+09,8.999999E+09,8.999999E+09,8.999999E+09]];
	LOCAL CONST Robtarget Tr_meulage_bavure_P8 :=[[3.41819189453125,59.48340234375,91.569953125],[0.284213845397937,-0.265440258548562,0.628829065072101,-0.673303769591659],[0,0,0,0],[8.999999E+09,8.999999E+09,8.999999E+09,8.999999E+09,8.999999E+09,8.999999E+09]];
	LOCAL CONST Robtarget Tr_meulage_bavure_P9 :=[[-0.958820983886719,55.14005859375,92.5973671875],[0.285807861531897,-0.266942308684276,0.628212680896572,-0.67261021229358],[0,0,0,0],[8.999999E+09,8.999999E+09,8.999999E+09,8.999999E+09,8.999999E+09,8.999999E+09]];
	LOCAL CONST Robtarget Tr_meulage_bavure_P10 :=[[-6.55028466796875,49.414171875,93.9323984375],[0.288322350056615,-0.269327080784598,0.627247398799099,-0.67148629674301],[0,0,0,0],[8.999999E+09,8.999999E+09,8.999999E+09,8.999999E+09,8.999999E+09,8.999999E+09]];
	LOCAL CONST Robtarget Tr_meulage_bavure_P11 :=[[-8.520876953125,47.44456640625,94.3967578125],[0.29141978931461,-0.272289487305219,0.62606789240698,-0.67005368113008],[0,0,0,0],[8.999999E+09,8.999999E+09,8.999999E+09,8.999999E+09,8.999999E+09,8.999999E+09]];
	LOCAL CONST Robtarget Tr_meulage_bavure_P12 :=[[-9.8624462890625,46.0195546875,94.723578125],[0.294369215143396,-0.275146476809444,0.624964034618918,-0.668626305875005],[0,0,0,0],[8.999999E+09,8.999999E+09,8.999999E+09,8.999999E+09,8.999999E+09,8.999999E+09]];
	LOCAL CONST Robtarget Tr_meulage_bavure_P13 :=[[-11.689984375,44.16079296875,95.1583125],[0.296268636909546,-0.277054979800622,0.624311920199916,-0.667607713592144],[0,0,0,0],[8.999999E+09,8.999999E+09,8.999999E+09,8.999999E+09,8.999999E+09,8.999999E+09]];
	LOCAL CONST Robtarget Tr_meulage_bavure_P14 :=[[-11.7441982421875,44.07610546875,95.1749609375],[0.29642432777975,-0.277366079829103,0.624411730781714,-0.667316016683807],[0,0,0,0],[8.999999E+09,8.999999E+09,8.999999E+09,8.999999E+09,8.999999E+09,8.999999E+09]];
	LOCAL CONST Robtarget Tr_meulage_bavure_P15 :=[[-14.0992275390625,41.6959140625,95.7332578125],[0.294687475657803,-0.275932746223752,0.625323368688705,-0.667825647773175],[0,0,0,0],[8.999999E+09,8.999999E+09,8.999999E+09,8.999999E+09,8.999999E+09,8.999999E+09]];
	LOCAL CONST Robtarget Tr_meulage_bavure_P16 :=[[-14.4200859375,41.392875,95.806625],[0.291523045570414,-0.273182110372919,0.626838877391853,-0.668923665498292],[0,0,0,0],[8.999999E+09,8.999999E+09,8.999999E+09,8.999999E+09,8.999999E+09,8.999999E+09]];
	LOCAL CONST Robtarget Tr_meulage_bavure_P17 :=[[-15.989626953125,39.8081171875,96.1785078125],[0.28777160038532,-0.269893857490973,0.628595285599939,-0.670233376236849],[0,0,0,0],[8.999999E+09,8.999999E+09,8.999999E+09,8.999999E+09,8.999999E+09,8.999999E+09]];
	LOCAL CONST Robtarget Tr_meulage_bavure_P18 :=[[-20.5275,35.3738203125,97.234953125],[0.284306583970974,-0.266879921516261,0.630230152784219,-0.671382773329649],[0,0,0,0],[8.999999E+09,8.999999E+09,8.999999E+09,8.999999E+09,8.999999E+09,8.999999E+09]];
	LOCAL CONST Robtarget Tr_meulage_bavure_P19 :=[[-21.675865234375,34.22190234375,97.5060859375],[0.281736631260211,-0.264703803449232,0.631499517747391,-0.672134455395994],[0,0,0,0],[8.999999E+09,8.999999E+09,8.999999E+09,8.999999E+09,8.999999E+09,8.999999E+09]];
	LOCAL CONST Robtarget Tr_meulage_bavure_P20 :=[[-25.820263671875,30.174119140625,98.470671875],[0.280280494877072,-0.263565603698652,0.632319207039449,-0.672419836967524],[0,0,0,0],[8.999999E+09,8.999999E+09,8.999999E+09,8.999999E+09,8.999999E+09,8.999999E+09]];
	LOCAL CONST Robtarget Tr_meulage_bavure_P21 :=[[-29.943333984375,25.966017578125,99.4533203125],[0.279831511777758,-0.263365067852669,0.632734307370033,-0.672294922134697],[0,0,0,0],[8.999999E+09,8.999999E+09,8.999999E+09,8.999999E+09,8.999999E+09,8.999999E+09]];
	LOCAL CONST Robtarget Tr_meulage_bavure_P22 :=[[-30.65425390625,25.273341796875,99.6185703125],[0.280098455209423,-0.263823147198514,0.632852238379101,-0.671893032238115],[0,0,0,0],[8.999999E+09,8.999999E+09,8.999999E+09,8.999999E+09,8.999999E+09,8.999999E+09]];
	LOCAL CONST Robtarget Tr_meulage_bavure_P23 :=[[-31.59001953125,24.25621875,99.8494765625],[0.280755004027766,-0.264628999192664,0.632794717727717,-0.671356064779009],[0,0,0,0],[8.999999E+09,8.999999E+09,8.999999E+09,8.999999E+09,8.999999E+09,8.999999E+09]];
	LOCAL CONST Robtarget Tr_meulage_bavure_P24 :=[[-33.03751171875,22.785212890625,100.1936484375],[0.281494324913843,-0.265490782989762,0.632678385129633,-0.670815660355766],[0,0,0,0],[8.999999E+09,8.999999E+09,8.999999E+09,8.999999E+09,8.999999E+09,8.999999E+09]];
	LOCAL CONST Robtarget Tr_meulage_bavure_P25 :=[[-35.58303125,20.01735546875,100.8218984375],[0.282069674309091,-0.266177353782537,0.632602905091275,-0.670372940711787],[0,0,0,0],[8.999999E+09,8.999999E+09,8.999999E+09,8.999999E+09,8.999999E+09,8.999999E+09]];
	LOCAL CONST Robtarget Tr_meulage_bavure_P26 :=[[-35.98186328125,19.596505859375,100.918703125],[0.28234267845556,-0.266560840783109,0.632627454835272,-0.670082407970981],[0,0,0,0],[8.999999E+09,8.999999E+09,8.999999E+09,8.999999E+09,8.999999E+09,8.999999E+09]];
	LOCAL CONST Robtarget Tr_meulage_bavure_P27 :=[[-35.99944140625,19.584302734375,100.9221640625],[0.282265557944378,-0.26659776528805,0.632774037575629,-0.669961792725529],[0,0,0,0],[8.999999E+09,8.999999E+09,8.999999E+09,8.999999E+09,8.999999E+09,8.999999E+09]];
	LOCAL CONST Robtarget Tr_meulage_bavure_P28 :=[[-36.72640234375,18.841884765625,101.0954765625],[0.281868959392986,-0.266325730096396,0.633040201901723,-0.669985520735756],[0,0,0,0],[8.999999E+09,8.999999E+09,8.999999E+09,8.999999E+09,8.999999E+09,8.999999E+09]];
	LOCAL CONST Robtarget Tr_meulage_bavure_P29 :=[[-40.45190234375,15.164779296875,101.967453125],[0.281268755948015,-0.265862992961441,0.633389182694683,-0.670091709504306],[0,0,0,0],[8.999999E+09,8.999999E+09,8.999999E+09,8.999999E+09,8.999999E+09,8.999999E+09]];
	LOCAL CONST Robtarget Tr_meulage_bavure_P30 :=[[-46.5366875,9.034759765625,103.4074296875],[0.280629008001166,-0.265374589995516,0.633766366094151,-0.670196896487001],[0,0,0,0],[8.999999E+09,8.999999E+09,8.999999E+09,8.999999E+09,8.999999E+09,8.999999E+09]];
	LOCAL CONST Robtarget Tr_meulage_bavure_P31 :=[[-47.9009765625,7.66512158203125,103.7296875],[0.280126846706262,-0.265044675438766,0.634119448740969,-0.670203547069407],[0,0,0,0],[8.999999E+09,8.999999E+09,8.999999E+09,8.999999E+09,8.999999E+09,8.999999E+09]];
	LOCAL CONST Robtarget Tr_meulage_bavure_P32 :=[[-49.00028515625,6.58895849609375,103.985859375],[0.279912301482713,-0.26502575630409,0.634400388606441,-0.670034774403607],[0,0,0,0],[8.999999E+09,8.999999E+09,8.999999E+09,8.999999E+09,8.999999E+09,8.999999E+09]];
	LOCAL CONST Robtarget Tr_meulage_bavure_P33 :=[[-56.24496875,-0.754955444335938,105.70609375],[0.280039190285508,-0.265387076054559,0.634606547332694,-0.669643399019154],[0,0,0,0],[8.999999E+09,8.999999E+09,8.999999E+09,8.999999E+09,8.999999E+09,8.999999E+09]];
	LOCAL CONST Robtarget Tr_meulage_bavure_P34 :=[[-56.44252734375,-0.940341125488281,105.751109375],[0.280436694311137,-0.266076323772035,0.634779618441978,-0.669039226370516],[0,0,0,0],[8.999999E+09,8.999999E+09,8.999999E+09,8.999999E+09,8.999999E+09,8.999999E+09]];
	LOCAL CONST Robtarget Tr_meulage_bavure_P35 :=[[-61.49255859375,-6.014634765625,106.9445234375],[0.28089986869357,-0.266914266221368,0.635014623407983,-0.668287712226899],[0,0,0,0],[8.999999E+09,8.999999E+09,8.999999E+09,8.999999E+09,8.999999E+09,8.999999E+09]];
	LOCAL CONST Robtarget Tr_meulage_bavure_P36 :=[[-62.0686875,-6.60664013671875,107.08234375],[0.281135980929385,-0.267639959443632,0.635445326692624,-0.66748831384556],[0,0,0,0],[8.999999E+09,8.999999E+09,8.999999E+09,8.999999E+09,8.999999E+09,8.999999E+09]];
	LOCAL CONST Robtarget Tr_meulage_bavure_P37 :=[[-62.15234765625,-6.68784228515625,107.10175],[0.280872409861467,-0.268002066607424,0.636191141596299,-0.666743138717722],[0,0,0,0],[8.999999E+09,8.999999E+09,8.999999E+09,8.999999E+09,8.999999E+09,8.999999E+09]];
	LOCAL CONST Robtarget Tr_meulage_bavure_P38 :=[[-62.4766171875,-7.02322021484375,107.17959375],[0.279952648313818,-0.267860150951519,0.637328446406798,-0.666100522169895],[0,0,0,0],[8.999999E+09,8.999999E+09,8.999999E+09,8.999999E+09,8.999999E+09,8.999999E+09]];
	LOCAL CONST Robtarget Tr_meulage_bavure_P39 :=[[-63.384140625,-7.966861328125,107.39809375],[0.278409568963992,-0.267250326223849,0.638854365642366,-0.665530220607765],[0,0,0,0],[8.999999E+09,8.999999E+09,8.999999E+09,8.999999E+09,8.999999E+09,8.999999E+09]];
	LOCAL CONST Robtarget Tr_meulage_bavure_P40 :=[[-76.2720078125,-21.096939453125,110.4666328125],[0.27647060340918,-0.2663891523062,0.64068105745596,-0.6649275205624],[0,0,0,0],[8.999999E+09,8.999999E+09,8.999999E+09,8.999999E+09,8.999999E+09,8.999999E+09]];
	LOCAL CONST Robtarget Tr_meulage_bavure_P41 :=[[-80.59846875,-25.452609375,111.490125],[0.274546255000979,-0.26567165495655,0.642647017176692,-0.664114249908467],[0,0,0,0],[8.999999E+09,8.999999E+09,8.999999E+09,8.999999E+09,8.999999E+09,8.999999E+09]];
	LOCAL CONST Robtarget Tr_meulage_bavure_P42 :=[[-83.3634140625,-28.0718984375,112.1233359375],[0.273144744796606,-0.265588810037895,0.644546334529159,-0.662883515421584],[0,0,0,0],[8.999999E+09,8.999999E+09,8.999999E+09,8.999999E+09,8.999999E+09,8.999999E+09]];
	LOCAL CONST Robtarget Tr_meulage_bavure_P43 :=[[-86.130109375,-30.768453125,112.7665546875],[0.272817776514206,-0.266688663135384,0.646156350621466,-0.661006496431355],[0,0,0,0],[8.999999E+09,8.999999E+09,8.999999E+09,8.999999E+09,8.999999E+09,8.999999E+09]];
	LOCAL CONST Robtarget Tr_meulage_bavure_P44 :=[[-86.8596484375,-31.48644140625,112.9370390625],[0.27428351230221,-0.269688662603679,0.647164415709515,-0.658190549295236],[0,0,0,0],[8.999999E+09,8.999999E+09,8.999999E+09,8.999999E+09,8.999999E+09,8.999999E+09]];
	LOCAL CONST Robtarget Tr_meulage_bavure_P45 :=[[-88.19725,-32.81711328125,113.2514453125],[0.278407617210333,-0.275468154571829,0.647155596433672,-0.65406125745272],[0,0,0,0],[8.999999E+09,8.999999E+09,8.999999E+09,8.999999E+09,8.999999E+09,8.999999E+09]];
	LOCAL CONST Robtarget Tr_meulage_bavure_P46 :=[[-91.98925,-36.439203125,114.12365625],[0.286353616651651,-0.285230997494903,0.645506962357269,-0.648047564494207],[0,0,0,0],[8.999999E+09,8.999999E+09,8.999999E+09,8.999999E+09,8.999999E+09,8.999999E+09]];
	LOCAL CONST Robtarget Tr_meulage_bavure_P47 :=[[-95.3056484375,-39.89283203125,114.922796875],[0.299650668113211,-0.300587306240852,0.641254795041416,-0.639256627859709],[0,0,0,0],[8.999999E+09,8.999999E+09,8.999999E+09,8.999999E+09,8.999999E+09,8.999999E+09]];
	LOCAL CONST Robtarget Tr_meulage_bavure_P48 :=[[-100.4908984375,-45.2673359375,116.169046875],[0.320051028593992,-0.323416808300398,0.632955064228461,-0.626367938094101],[0,0,0,0],[8.999999E+09,8.999999E+09,8.999999E+09,8.999999E+09,8.999999E+09,8.999999E+09]];
	LOCAL CONST Robtarget Tr_meulage_bavure_P49 :=[[-103.1467109375,-47.98748046875,116.8032109375],[0.349083003066893,-0.355430902110319,0.618610109095904,-0.607561901141931],[0,0,0,0],[8.999999E+09,8.999999E+09,8.999999E+09,8.999999E+09,8.999999E+09,8.999999E+09]];
	LOCAL CONST Robtarget Tr_meulage_bavure_P50 :=[[-104.90665625,-50.2904921875,117.2870546875],[0.387058512056147,-0.397136430194387,0.595929379738561,-0.580806799565702],[0,0,0,0],[8.999999E+09,8.999999E+09,8.999999E+09,8.999999E+09,8.999999E+09,8.999999E+09]];
	LOCAL CONST Robtarget Tr_meulage_bavure_P51 :=[[-105.5893203125,-51.99621875,117.57796875],[0.43184428563275,-0.44652973010744,0.563316451820981,-0.544790132256759],[0,0,0,0],[8.999999E+09,8.999999E+09,8.999999E+09,8.999999E+09,8.999999E+09,8.999999E+09]];
	LOCAL CONST Robtarget Tr_meulage_bavure_P52 :=[[-106.2798515625,-54.09439453125,117.9196015625],[0.478392482158397,-0.498481197686526,0.52160530549503,-0.500584691982057],[0,0,0,0],[8.999999E+09,8.999999E+09,8.999999E+09,8.999999E+09,8.999999E+09,8.999999E+09]];
	LOCAL CONST Robtarget Tr_meulage_bavure_P53 :=[[-106.24278125,-54.8323671875,118.0093515625],[0.520658622167301,-0.546637683470221,0.474882966311317,-0.452314061776242],[0,0,0,0],[8.999999E+09,8.999999E+09,8.999999E+09,8.999999E+09,8.999999E+09,8.999999E+09]];
	LOCAL CONST Robtarget Tr_meulage_bavure_P54 :=[[-105.2187578125,-57.02176953125,118.1763203125],[0.554709056689723,-0.586678986818574,0.42871377759736,-0.405351854257668],[0,0,0,0],[8.999999E+09,8.999999E+09,8.999999E+09,8.999999E+09,8.999999E+09,8.999999E+09]];
	LOCAL CONST Robtarget Tr_meulage_bavure_P55 :=[[-104.978359375,-57.656765625,118.2308984375],[0.579801101572751,-0.617550876730381,0.387462675636133,-0.363777778669137],[0,0,0,0],[8.999999E+09,8.999999E+09,8.999999E+09,8.999999E+09,8.999999E+09,8.999999E+09]];
	LOCAL CONST Robtarget Tr_meulage_bavure_P56 :=[[-104.8231328125,-57.89610546875,118.2444453125],[0.597111227807004,-0.640236934194449,0.353422853377421,-0.329616650718174],[0,0,0,0],[8.999999E+09,8.999999E+09,8.999999E+09,8.999999E+09,8.999999E+09,8.999999E+09]];
	LOCAL CONST Robtarget Tr_meulage_bavure_P57 :=[[-103.4312578125,-59.53333203125,118.3012890625],[0.608331665190778,-0.656340290957888,0.327298218171311,-0.303357683227926],[0,0,0,0],[8.999999E+09,8.999999E+09,8.999999E+09,8.999999E+09,8.999999E+09,8.999999E+09]];
	LOCAL CONST Robtarget Tr_meulage_bavure_P58 :=[[-102.9890546875,-59.9969296875,118.31215625],[0.615011742863901,-0.667368044766304,0.308835564102726,-0.284606822317489],[0,0,0,0],[8.999999E+09,8.999999E+09,8.999999E+09,8.999999E+09,8.999999E+09,8.999999E+09]];
	LOCAL CONST Robtarget Tr_meulage_bavure_P59 :=[[-100.397296875,-62.29012109375,118.3220078125],[0.61845408506239,-0.674611894552726,0.297063956793492,-0.272334981175422],[0,0,0,0],[8.999999E+09,8.999999E+09,8.999999E+09,8.999999E+09,8.999999E+09,8.999999E+09]];
	LOCAL CONST Robtarget Tr_meulage_bavure_P60 :=[[-95.87471875,-66.59021875,118.377125],[0.619715785437852,-0.67915851952747,0.29053891952191,-0.265109763825179],[0,0,0,0],[8.999999E+09,8.999999E+09,8.999999E+09,8.999999E+09,8.999999E+09,8.999999E+09]];
	LOCAL CONST Robtarget Tr_meulage_bavure_P61 :=[[-91.1348359375,-71.514203125,118.48790625],[0.619665131833267,-0.681907379741001,0.287600458897685,-0.261349241220753],[0,0,0,0],[8.999999E+09,8.999999E+09,8.999999E+09,8.999999E+09,8.999999E+09,8.999999E+09]];
	LOCAL CONST Robtarget Tr_meulage_bavure_P62 :=[[-90.9986953125,-71.6591328125,118.4915390625],[0.618955368390622,-0.683568560663652,0.286737509367227,-0.259634118587161],[0,0,0,0],[8.999999E+09,8.999999E+09,8.999999E+09,8.999999E+09,8.999999E+09,8.999999E+09]];
	LOCAL CONST Robtarget Tr_meulage_bavure_P63 :=[[-90.9642265625,-71.6925,118.49203125],[0.617997226649173,-0.684607270695193,0.286906891985544,-0.258991791561826],[0,0,0,0],[8.999999E+09,8.999999E+09,8.999999E+09,8.999999E+09,8.999999E+09,8.999999E+09]];
	LOCAL CONST Robtarget Tr_meulage_bavure_P64 :=[[-88.8031953125,-73.8572734375,118.5323515625],[0.617005567161032,-0.685270329347304,0.287542199192477,-0.25889802913905],[0,0,0,0],[8.999999E+09,8.999999E+09,8.999999E+09,8.999999E+09,8.999999E+09,8.999999E+09]];
	LOCAL CONST Robtarget Tr_meulage_bavure_P65 :=[[-86.8116875,-75.7042578125,118.550703125],[0.616040099710545,-0.685652060361261,0.288455885707406,-0.259169924319423],[0,0,0,0],[8.999999E+09,8.999999E+09,8.999999E+09,8.999999E+09,8.999999E+09,8.999999E+09]];
	LOCAL CONST Robtarget Tr_meulage_bavure_P66 :=[[-83.74115625,-78.588890625,118.5836953125],[0.615091377406664,-0.685776540747927,0.289633396252619,-0.259779963382383],[0,0,0,0],[8.999999E+09,8.999999E+09,8.999999E+09,8.999999E+09,8.999999E+09,8.999999E+09]];
	LOCAL CONST Robtarget Tr_meulage_bavure_P67 :=[[-79.935671875,-82.4907265625,118.666109375],[0.614112759090037,-0.685622234066547,0.29116080750434,-0.260793127689057],[0,0,0,0],[8.999999E+09,8.999999E+09,8.999999E+09,8.999999E+09,8.999999E+09,8.999999E+09]];
	LOCAL CONST Robtarget Tr_meulage_bavure_P68 :=[[-78.99553125,-83.4622421875,118.6874296875],[0.613073056053647,-0.685160330665169,0.293107232236333,-0.262268754590771],[0,0,0,0],[8.999999E+09,8.999999E+09,8.999999E+09,8.999999E+09,8.999999E+09,8.999999E+09]];
	LOCAL CONST Robtarget Tr_meulage_bavure_P69 :=[[-73.666015625,-88.6637890625,118.7694296875],[0.611906120595634,-0.684416402837857,0.2955251198127,-0.264215803205976],[0,0,0,0],[8.999999E+09,8.999999E+09,8.999999E+09,8.999999E+09,8.999999E+09,8.999999E+09]];
	LOCAL CONST Robtarget Tr_meulage_bavure_P70 :=[[-72.0848671875,-90.22696875,118.7963046875],[0.610630083679486,-0.683415806300978,0.298348926725825,-0.266573919439087],[0,0,0,0],[8.999999E+09,8.999999E+09,8.999999E+09,8.999999E+09,8.999999E+09,8.999999E+09]];
	LOCAL CONST Robtarget Tr_meulage_bavure_P71 :=[[-69.2236953125,-93.204796875,118.8638828125],[0.609350542411906,-0.682273292790736,0.301300445916409,-0.269096844458229],[0,0,0,0],[8.999999E+09,8.999999E+09,8.999999E+09,8.999999E+09,8.999999E+09,8.999999E+09]];
	LOCAL CONST Robtarget Tr_meulage_bavure_P72 :=[[-64.37560546875,-97.9457890625,118.93965625],[0.608228774854949,-0.68123250638563,0.303903048854299,-0.271335523990247],[0,0,0,0],[8.999999E+09,8.999999E+09,8.999999E+09,8.999999E+09,8.999999E+09,8.999999E+09]];
	LOCAL CONST Robtarget Tr_meulage_bavure_P73 :=[[-55.29626171875,-106.8903671875,119.0899375],[0.607495640747576,-0.680586127214236,0.305555353140486,-0.272740712185425],[0,0,0,0],[8.999999E+09,8.999999E+09,8.999999E+09,8.999999E+09,8.999999E+09,8.999999E+09]];
	LOCAL CONST Robtarget Tr_meulage_bavure_P74 :=[[-53.3141875,-108.8420546875,119.1226171875],[0.607365723860621,-0.680561439913334,0.305753726546202,-0.272869314298008],[0,0,0,0],[8.999999E+09,8.999999E+09,8.999999E+09,8.999999E+09,8.999999E+09,8.999999E+09]];
	LOCAL CONST Robtarget Tr_meulage_bavure_P75 :=[[-52.98756640625,-109.259328125,119.1401640625],[0.607874701514068,-0.681260619156945,0.304346107600989,-0.271561710911546],[0,0,0,0],[8.999999E+09,8.999999E+09,8.999999E+09,8.999999E+09,8.999999E+09,8.999999E+09]];
	LOCAL CONST Robtarget Tr_meulage_bavure_P76 :=[[-48.425359375,-113.83596875,119.2261171875],[0.608903346403116,-0.682538270929206,0.301619565671816,-0.269079655604063],[0,0,0,0],[8.999999E+09,8.999999E+09,8.999999E+09,8.999999E+09,8.999999E+09,8.999999E+09]];
	LOCAL CONST Robtarget Tr_meulage_bavure_P77 :=[[-45.45498828125,-116.83284375,119.28425],[0.610182082227783,-0.684113324447558,0.298201329916801,-0.2659750978519],[0,0,0,0],[8.999999E+09,8.999999E+09,8.999999E+09,8.999999E+09,8.999999E+09,8.999999E+09]];
	LOCAL CONST Robtarget Tr_meulage_bavure_P78 :=[[-38.87232421875,-123.290171875,119.3896953125],[0.611433048829487,-0.685658091047738,0.294805761477729,-0.262891939738338],[0,0,0,0],[8.999999E+09,8.999999E+09,8.999999E+09,8.999999E+09,8.999999E+09,8.999999E+09]];
	LOCAL CONST Robtarget Tr_meulage_bavure_P79 :=[[-36.155046875,-125.9686953125,119.4348671875],[0.612443420773068,-0.686949238146479,0.291979109920202,-0.260311351907598],[0,0,0,0],[8.999999E+09,8.999999E+09,8.999999E+09,8.999999E+09,8.999999E+09,8.999999E+09]];
	LOCAL CONST Robtarget Tr_meulage_bavure_P80 :=[[-32.331330078125,-129.7638203125,119.501734375],[0.613108197372345,-0.687922093495886,0.289960777628354,-0.258426544751564],[0,0,0,0],[8.999999E+09,8.999999E+09,8.999999E+09,8.999999E+09,8.999999E+09,8.999999E+09]];
	LOCAL CONST Robtarget Tr_meulage_bavure_P81 :=[[-29.685912109375,-132.419078125,119.551765625],[0.613486045778431,-0.688585830139755,0.288678819439904,-0.257194411628],[0,0,0,0],[8.999999E+09,8.999999E+09,8.999999E+09,8.999999E+09,8.999999E+09,8.999999E+09]];
	LOCAL CONST Robtarget Tr_meulage_bavure_P82 :=[[-28.723173828125,-133.389984375,119.570546875],[0.613674346755665,-0.689018396300321,0.287920096689541,-0.256436080955912],[0,0,0,0],[8.999999E+09,8.999999E+09,8.999999E+09,8.999999E+09,8.999999E+09,8.999999E+09]];
	LOCAL CONST Robtarget Tr_meulage_bavure_P83 :=[[-28.204634765625,-133.882515625,119.5768046875],[0.613725445895417,-0.689319597240136,0.28750193007431,-0.255973065232876],[0,0,0,0],[8.999999E+09,8.999999E+09,8.999999E+09,8.999999E+09,8.999999E+09,8.999999E+09]];
	LOCAL CONST Robtarget Tr_meulage_bavure_P84 :=[[-22.6324140625,-139.494703125,119.684625],[0.613690126247506,-0.689519970118323,0.287320097384191,-0.255722117528941],[0,0,0,0],[8.999999E+09,8.999999E+09,8.999999E+09,8.999999E+09,8.999999E+09,8.999999E+09]];
	LOCAL CONST Robtarget Tr_meulage_bavure_P85 :=[[-18.860220703125,-143.12709375,119.7364140625],[0.613574239444196,-0.68961398483375,0.287373594027721,-0.255686569979308],[0,0,0,0],[8.999999E+09,8.999999E+09,8.999999E+09,8.999999E+09,8.999999E+09,8.999999E+09]];
	LOCAL CONST Robtarget Tr_meulage_bavure_P86 :=[[-16.972771484375,-144.9145625,119.7585078125],[0.613403067694079,-0.68955632792265,0.287679472474156,-0.255908710837117],[0,0,0,0],[8.999999E+09,8.999999E+09,8.999999E+09,8.999999E+09,8.999999E+09,8.999999E+09]];
	LOCAL CONST Robtarget Tr_meulage_bavure_P87 :=[[-15.484251953125,-146.432765625,119.7897265625],[0.613171082772722,-0.689359716705175,0.288229952556613,-0.256374528151105],[0,0,0,0],[8.999999E+09,8.999999E+09,8.999999E+09,8.999999E+09,8.999999E+09,8.999999E+09]];
	LOCAL CONST Robtarget Tr_meulage_bavure_P88 :=[[-9.040421875,-152.685140625,119.884203125],[0.612930383981775,-0.689053922145458,0.28891665036951,-0.256998455067686],[0,0,0,0],[8.999999E+09,8.999999E+09,8.999999E+09,8.999999E+09,8.999999E+09,8.999999E+09]];
	LOCAL CONST Robtarget Tr_meulage_bavure_P89 :=[[-8.2058798828125,-153.506125,119.8978671875],[0.612780710859617,-0.688694971118761,0.289535537613749,-0.257620281835163],[0,0,0,0],[8.999999E+09,8.999999E+09,8.999999E+09,8.999999E+09,8.999999E+09,8.999999E+09]];
	LOCAL CONST Robtarget Tr_meulage_bavure_P90 :=[[-7.8719853515625,-153.849484375,119.905234375],[0.612810067539707,-0.688370477722823,0.289864753634522,-0.258047149029067],[0,0,0,0],[8.999999E+09,8.999999E+09,8.999999E+09,8.999999E+09,8.999999E+09,8.999999E+09]];
	LOCAL CONST Robtarget Tr_meulage_bavure_P91 :=[[-7.72273291015625,-153.990640625,119.906953125],[0.613095284935195,-0.688133569717675,0.289738328538041,-0.258143492642799],[0,0,0,0],[8.999999E+09,8.999999E+09,8.999999E+09,8.999999E+09,8.999999E+09,8.999999E+09]];
	LOCAL CONST Robtarget Tr_meulage_bavure_P92 :=[[-6.77853662109375,-154.94340625,119.925453125],[0.613661359849827,-0.687992047900235,0.289112701483239,-0.25787695378681],[0,0,0,0],[8.999999E+09,8.999999E+09,8.999999E+09,8.999999E+09,8.999999E+09,8.999999E+09]];
	LOCAL CONST Robtarget Tr_meulage_bavure_P93 :=[[-0.0936267852783203,-161.81665625,120.072640625],[0.614468375622735,-0.68790549321701,0.288087559443509,-0.257332869752978],[0,0,0,0],[8.999999E+09,8.999999E+09,8.999999E+09,8.999999E+09,8.999999E+09,8.999999E+09]];
	LOCAL CONST Robtarget Tr_meulage_bavure_P94 :=[[3.39895751953125,-165.264125,120.1313046875],[0.615472438752333,-0.687734461159857,0.286881043121286,-0.256737716681948],[0,0,0,0],[8.999999E+09,8.999999E+09,8.999999E+09,8.999999E+09,8.999999E+09,8.999999E+09]];
	LOCAL CONST Robtarget Tr_meulage_bavure_P95 :=[[5.38841845703125,-167.237015625,120.165875],[0.616516596930508,-0.687389243392371,0.285814682562872,-0.256346018126229],[0,0,0,0],[8.999999E+09,8.999999E+09,8.999999E+09,8.999999E+09,8.999999E+09,8.999999E+09]];
	LOCAL CONST Robtarget Tr_meulage_bavure_P96 :=[[7.4032607421875,-169.200078125,120.1964453125],[0.617562542095519,-0.686789438449565,0.285035037042871,-0.256304119148758],[0,0,0,0],[8.999999E+09,8.999999E+09,8.999999E+09,8.999999E+09,8.999999E+09,8.999999E+09]];
	LOCAL CONST Robtarget Tr_meulage_bavure_P97 :=[[10.77801171875,-172.5233125,120.252125],[0.618666265666939,-0.68597971679647,0.284411723385949,-0.256503121755259],[0,0,0,0],[8.999999E+09,8.999999E+09,8.999999E+09,8.999999E+09,8.999999E+09,8.999999E+09]];
	LOCAL CONST Robtarget Tr_meulage_bavure_P98 :=[[12.067623046875,-173.68325,120.259421875],[0.620055740895095,-0.685255559787293,0.283284551549278,-0.256330955635801],[0,0,0,0],[8.999999E+09,8.999999E+09,8.999999E+09,8.999999E+09,8.999999E+09,8.999999E+09]];
	LOCAL CONST Robtarget Tr_meulage_bavure_P99 :=[[14.82609375,-176.339125,120.29725],[0.622229286021663,-0.685151386473555,0.280329669070542,-0.254585093572142],[0,0,0,0],[8.999999E+09,8.999999E+09,8.999999E+09,8.999999E+09,8.999999E+09,8.999999E+09]];
	LOCAL CONST Robtarget Tr_meulage_bavure_P100 :=[[17.412205078125,-179.12378125,120.37015625],[0.625828056922003,-0.686388449231128,0.273722535272547,-0.249571860623924],[0,0,0,0],[8.999999E+09,8.999999E+09,8.999999E+09,8.999999E+09,8.999999E+09,8.999999E+09]];
	LOCAL CONST Robtarget Tr_meulage_bavure_P101 :=[[18.366267578125,-180.13265625,120.39471875],[0.631479223827229,-0.689635527832779,0.261416009669098,-0.239371047777401],[0,0,0,0],[8.999999E+09,8.999999E+09,8.999999E+09,8.999999E+09,8.999999E+09,8.999999E+09]];
	LOCAL CONST Robtarget Tr_meulage_bavure_P102 :=[[19.04490625,-180.822921875,120.408703125],[0.639381742860876,-0.695131202577719,0.241857333520494,-0.222460397197791],[0,0,0,0],[8.999999E+09,8.999999E+09,8.999999E+09,8.999999E+09,8.999999E+09,8.999999E+09]];
	LOCAL CONST Robtarget Tr_meulage_bavure_P103 :=[[19.53789453125,-181.3329375,120.4199609375],[0.649124998115778,-0.702393161264679,0.214467459869452,-0.198202655095604],[0,0,0,0],[8.999999E+09,8.999999E+09,8.999999E+09,8.999999E+09,8.999999E+09,8.999999E+09]];
	LOCAL CONST Robtarget Tr_meulage_bavure_P104 :=[[22.807076171875,-183.76065625,120.3733125],[0.659726691057129,-0.710326829452778,0.179773331063511,-0.166967176129636],[0,0,0,0],[8.999999E+09,8.999999E+09,8.999999E+09,8.999999E+09,8.999999E+09,8.999999E+09]];
	LOCAL CONST Robtarget Tr_meulage_bavure_P105 :=[[22.9763828125,-184.16425,120.406203125],[0.669990771433447,-0.717662142479234,0.138832674476175,-0.129610585771079],[0,0,0,0],[8.999999E+09,8.999999E+09,8.999999E+09,8.999999E+09,8.999999E+09,8.999999E+09]];
	LOCAL CONST Robtarget Tr_meulage_bavure_P106 :=[[24.207759765625,-184.914078125,120.3677109375],[0.678838671189368,-0.723283783675044,0.0923428541696716,-0.0866684720897004],[0,0,0,0],[8.999999E+09,8.999999E+09,8.999999E+09,8.999999E+09,8.999999E+09,8.999999E+09]];
	LOCAL CONST Robtarget Tr_meulage_bavure_P107 :=[[24.675912109375,-185.08234375,120.3382421875],[0.685271184352911,-0.726136649213437,0.040681748268599,-0.0383922638359704],[0,0,0,0],[8.999999E+09,8.999999E+09,8.999999E+09,8.999999E+09,8.999999E+09,8.999999E+09]];
	LOCAL CONST Robtarget Tr_meulage_bavure_P108 :=[[25.178181640625,-185.031484375,120.2772109375],[0.68824676976644,-0.725181174286762,-0.0150172429677993,0.0142523955803886],[0,0,0,0],[8.999999E+09,8.999999E+09,8.999999E+09,8.999999E+09,8.999999E+09,8.999999E+09]];
	LOCAL CONST Robtarget Tr_meulage_bavure_P109 :=[[27.59812890625,-185.296984375,120.0480625],[0.687099401305229,-0.719772153260911,-0.07168835947325,0.068434196365428],[0,0,0,0],[8.999999E+09,8.999999E+09,8.999999E+09,8.999999E+09,8.999999E+09,8.999999E+09]];
	LOCAL CONST Robtarget Tr_meulage_bavure_P110 :=[[29.19956640625,-185.09603125,119.8485546875],[0.682211877130918,-0.710426946525669,-0.124681150623313,0.119729357431545],[0,0,0,0],[8.999999E+09,8.999999E+09,8.999999E+09,8.999999E+09,8.999999E+09,8.999999E+09]];
	LOCAL CONST Robtarget Tr_meulage_bavure_P111 :=[[31.029787109375,-184.009828125,119.5116953125],[0.675185033947332,-0.698843380961394,-0.169797122581008,0.164048882907501],[0,0,0,0],[8.999999E+09,8.999999E+09,8.999999E+09,8.999999E+09,8.999999E+09,8.999999E+09]];
	LOCAL CONST Robtarget Tr_meulage_bavure_P112 :=[[32.1835703125,-183.372921875,119.305421875],[0.667954424264887,-0.687094622151526,-0.204995752572266,0.199285244668904],[0,0,0,0],[8.999999E+09,8.999999E+09,8.999999E+09,8.999999E+09,8.999999E+09,8.999999E+09]];
	LOCAL CONST Robtarget Tr_meulage_bavure_P113 :=[[33.84471875,-182.004859375,118.951125],[0.661944814227286,-0.676671275637231,-0.230468895433345,0.225453178914869],[0,0,0,0],[8.999999E+09,8.999999E+09,8.999999E+09,8.999999E+09,8.999999E+09,8.999999E+09]];
	LOCAL CONST Robtarget Tr_meulage_bavure_P114 :=[[34.00274609375,-181.870828125,118.916921875],[0.657826823046138,-0.668174824387936,-0.247680927205643,0.243845100901637],[0,0,0,0],[8.999999E+09,8.999999E+09,8.999999E+09,8.999999E+09,8.999999E+09,8.999999E+09]];
	LOCAL CONST Robtarget Tr_meulage_bavure_P115 :=[[39.5016875,-176.327890625,117.6151953125],[0.655548129122649,-0.661618300066037,-0.258591636215594,0.25621912711752],[0,0,0,0],[8.999999E+09,8.999999E+09,8.999999E+09,8.999999E+09,8.999999E+09,8.999999E+09]];
	LOCAL CONST Robtarget Tr_meulage_bavure_P116 :=[[40.33432421875,-175.45490625,117.4138046875],[0.654776675905897,-0.656613131843128,-0.265065239898854,0.264323889155229],[0,0,0,0],[8.999999E+09,8.999999E+09,8.999999E+09,8.999999E+09,8.999999E+09,8.999999E+09]];
	LOCAL CONST Robtarget Tr_meulage_bavure_P117 :=[[41.20657421875,-174.572265625,117.206890625],[0.655087932799514,-0.652735892848978,-0.268584106177654,0.269551910391778],[0,0,0,0],[8.999999E+09,8.999999E+09,8.999999E+09,8.999999E+09,8.999999E+09,8.999999E+09]];
	LOCAL CONST Robtarget Tr_meulage_bavure_P118 :=[[45.88188671875,-169.855765625,116.0996484375],[0.656124129022538,-0.649653813713489,-0.270175687008762,0.2728665384236],[0,0,0,0],[8.999999E+09,8.999999E+09,8.999999E+09,8.999999E+09,8.999999E+09,8.999999E+09]];
	LOCAL CONST Robtarget Tr_meulage_bavure_P119 :=[[49.67359375,-165.997140625,115.1974140625],[0.657670622391638,-0.647141147236999,-0.270442477666444,0.274842781002905],[0,0,0,0],[8.999999E+09,8.999999E+09,8.999999E+09,8.999999E+09,8.999999E+09,8.999999E+09]];
	LOCAL CONST Robtarget Tr_meulage_bavure_P120 :=[[50.97828515625,-164.7330625,114.895046875],[0.659604795971586,-0.645133412066269,-0.2696531788125,0.27570193492852],[0,0,0,0],[8.999999E+09,8.999999E+09,8.999999E+09,8.999999E+09,8.999999E+09,8.999999E+09]];
	LOCAL CONST Robtarget Tr_meulage_bavure_P121 :=[[51.62255859375,-164.014359375,114.733734375],[0.661834879023717,-0.643564449235236,-0.268013981447556,0.27562274640682],[0,0,0,0],[8.999999E+09,8.999999E+09,8.999999E+09,8.999999E+09,8.999999E+09,8.999999E+09]];
	LOCAL CONST Robtarget Tr_meulage_bavure_P122 :=[[53.6879921875,-162.00471875,114.253984375],[0.664234688564857,-0.642295867768708,-0.26583658230741,0.274916729686473],[0,0,0,0],[8.999999E+09,8.999999E+09,8.999999E+09,8.999999E+09,8.999999E+09,8.999999E+09]];
	LOCAL CONST Robtarget Tr_meulage_bavure_P123 :=[[59.7717109375,-156.043515625,112.835578125],[0.666591696990679,-0.641179208047342,-0.263561465364535,0.274007457281309],[0,0,0,0],[8.999999E+09,8.999999E+09,8.999999E+09,8.999999E+09,8.999999E+09,8.999999E+09]];
	LOCAL CONST Robtarget Tr_meulage_bavure_P124 :=[[62.14263671875,-153.60746875,112.268453125],[0.668691326475886,-0.640023673442931,-0.26167730425452,0.273398236582871],[0,0,0,0],[8.999999E+09,8.999999E+09,8.999999E+09,8.999999E+09,8.999999E+09,8.999999E+09]];
	LOCAL CONST Robtarget Tr_meulage_bavure_P125 :=[[64.88026171875,-150.886359375,111.6252734375],[0.670350266572393,-0.638687988108945,-0.26058465114333,0.273502858376614],[0,0,0,0],[8.999999E+09,8.999999E+09,8.999999E+09,8.999999E+09,8.999999E+09,8.999999E+09]];
	LOCAL CONST Robtarget Tr_meulage_bavure_P126 :=[[67.7771640625,-148.082578125,110.9542890625],[0.6715237348866,-0.637100164622218,-0.260415826682118,0.274486522320793],[0,0,0,0],[8.999999E+09,8.999999E+09,8.999999E+09,8.999999E+09,8.999999E+09,8.999999E+09]];
	LOCAL CONST Robtarget Tr_meulage_bavure_P127 :=[[70.4065546875,-145.477859375,110.33765625],[0.672274375948197,-0.635337045096306,-0.261000804694258,0.276174912909749],[0,0,0,0],[8.999999E+09,8.999999E+09,8.999999E+09,8.999999E+09,8.999999E+09,8.999999E+09]];
	LOCAL CONST Robtarget Tr_meulage_bavure_P128 :=[[72.874484375,-143.13878125,109.7723203125],[0.672746805309996,-0.633586970070095,-0.261949548877301,0.27813975110647],[0,0,0,0],[8.999999E+09,8.999999E+09,8.999999E+09,8.999999E+09,8.999999E+09,8.999999E+09]];
	LOCAL CONST Robtarget Tr_meulage_bavure_P129 :=[[78.821390625,-137.26746875,108.3801953125],[0.673176445179979,-0.632007327080715,-0.262783781220594,0.279901583594204],[0,0,0,0],[8.999999E+09,8.999999E+09,8.999999E+09,8.999999E+09,8.999999E+09,8.999999E+09]];
	LOCAL CONST Robtarget Tr_meulage_bavure_P130 :=[[79.707203125,-136.411609375,108.1752109375],[0.67373038942611,-0.630733387902798,-0.263153430506957,0.281092560842192],[0,0,0,0],[8.999999E+09,8.999999E+09,8.999999E+09,8.999999E+09,8.999999E+09,8.999999E+09]];
	LOCAL CONST Robtarget Tr_meulage_bavure_P131 :=[[81.46096875,-134.633625,107.7587578125],[0.674464969554322,-0.629803777952747,-0.26295433392988,0.281601179663771],[0,0,0,0],[8.999999E+09,8.999999E+09,8.999999E+09,8.999999E+09,8.999999E+09,8.999999E+09]];
	LOCAL CONST Robtarget Tr_meulage_bavure_P132 :=[[83.962171875,-131.9999375,107.1523671875],[0.675341382633046,-0.629144885169229,-0.262311865358335,0.281572753761642],[0,0,0,0],[8.999999E+09,8.999999E+09,8.999999E+09,8.999999E+09,8.999999E+09,8.999999E+09]];
	LOCAL CONST Robtarget Tr_meulage_bavure_P133 :=[[86.468421875,-129.4117734375,106.55121875],[0.676253255418065,-0.628642273838876,-0.261478427791629,0.28128181220757],[0,0,0,0],[8.999999E+09,8.999999E+09,8.999999E+09,8.999999E+09,8.999999E+09,8.999999E+09]];
	LOCAL CONST Robtarget Tr_meulage_bavure_P134 :=[[88.824828125,-126.9921484375,105.9877578125],[0.677139812905977,-0.628166029273746,-0.260655269495037,0.2809767675958],[0,0,0,0],[8.999999E+09,8.999999E+09,8.999999E+09,8.999999E+09,8.999999E+09,8.999999E+09]];
	LOCAL CONST Robtarget Tr_meulage_bavure_P135 :=[[91.127875,-124.631359375,105.437578125],[0.677968262960954,-0.627683776626322,-0.259917651460795,0.280739960527404],[0,0,0,0],[8.999999E+09,8.999999E+09,8.999999E+09,8.999999E+09,8.999999E+09,8.999999E+09]];
	LOCAL CONST Robtarget Tr_meulage_bavure_P136 :=[[91.850140625,-124.00771875,105.2798671875],[0.678782179297892,-0.627185483814133,-0.259213309756743,0.280538022388038],[0,0,0,0],[8.999999E+09,8.999999E+09,8.999999E+09,8.999999E+09,8.999999E+09,8.999999E+09]];
	LOCAL CONST Robtarget Tr_meulage_bavure_P137 :=[[93.0625234375,-122.7440703125,104.9875859375],[0.679654976161815,-0.626689876555652,-0.258421821886639,0.28026250904096],[0,0,0,0],[8.999999E+09,8.999999E+09,8.999999E+09,8.999999E+09,8.999999E+09,8.999999E+09]];
	LOCAL CONST Robtarget Tr_meulage_bavure_P138 :=[[95.629703125,-120.1096640625,104.3739375],[0.680611620517295,-0.626235126194352,-0.257473397171851,0.279830017128169],[0,0,0,0],[8.999999E+09,8.999999E+09,8.999999E+09,8.999999E+09,8.999999E+09,8.999999E+09]];
	LOCAL CONST Robtarget Tr_meulage_bavure_P139 :=[[96.5507109375,-119.15375,104.1524140625],[0.681644585494143,-0.625820510394285,-0.256378557812666,0.279247887960236],[0,0,0,0],[8.999999E+09,8.999999E+09,8.999999E+09,8.999999E+09,8.999999E+09,8.999999E+09]];
	LOCAL CONST Robtarget Tr_meulage_bavure_P140 :=[[102.7818046875,-112.9090625,102.6819765625],[0.682742785545597,-0.625388323350711,-0.255203811534816,0.278608593514501],[0,0,0,0],[8.999999E+09,8.999999E+09,8.999999E+09,8.999999E+09,8.999999E+09,8.999999E+09]];
	LOCAL CONST Robtarget Tr_meulage_bavure_P141 :=[[102.8521796875,-112.839515625,102.6654921875],[0.683850813564494,-0.624926155185293,-0.254038756674767,0.277992221940913],[0,0,0,0],[8.999999E+09,8.999999E+09,8.999999E+09,8.999999E+09,8.999999E+09,8.999999E+09]];
	LOCAL CONST Robtarget Tr_meulage_bavure_P142 :=[[102.874859375,-112.8187890625,102.660390625],[0.684949316985706,-0.624434745548718,-0.252910444396717,0.277420238676593],[0,0,0,0],[8.999999E+09,8.999999E+09,8.999999E+09,8.999999E+09,8.999999E+09,8.999999E+09]];
	LOCAL CONST Robtarget Tr_meulage_bavure_P143 :=[[102.883546875,-112.808328125,102.6581171875],[0.686044756307933,-0.623964049259895,-0.251764807887635,0.276813906953545],[0,0,0,0],[8.999999E+09,8.999999E+09,8.999999E+09,8.999999E+09,8.999999E+09,8.999999E+09]];
	LOCAL CONST Robtarget Tr_meulage_bavure_P144 :=[[107.5908515625,-108.2330390625,101.5653515625],[0.687191725938432,-0.623595823543057,-0.250449325152078,0.275990790049748],[0,0,0,0],[8.999999E+09,8.999999E+09,8.999999E+09,8.999999E+09,8.999999E+09,8.999999E+09]];
	LOCAL CONST Robtarget Tr_meulage_bavure_P145 :=[[108.366875,-107.3240234375,101.3655390625],[0.68844874229726,-0.623430272019133,-0.248786666103338,0.274732997524244],[0,0,0,0],[8.999999E+09,8.999999E+09,8.999999E+09,8.999999E+09,8.999999E+09,8.999999E+09]];
	LOCAL CONST Robtarget Tr_meulage_bavure_P146 :=[[111.11371875,-104.544515625,100.7139375],[0.689841427882166,-0.623533535234899,-0.246673156033977,0.27290490817719],[0,0,0,0],[8.999999E+09,8.999999E+09,8.999999E+09,8.999999E+09,8.999999E+09,8.999999E+09]];
	LOCAL CONST Robtarget Tr_meulage_bavure_P147 :=[[111.905390625,-103.76434375,100.5287890625],[0.691312775698093,-0.623907733047199,-0.244179044323363,0.270559385558572],[0,0,0,0],[8.999999E+09,8.999999E+09,8.999999E+09,8.999999E+09,8.999999E+09,8.999999E+09]];
	LOCAL CONST Robtarget Tr_meulage_bavure_P148 :=[[114.3721640625,-101.0999921875,99.92225],[0.69272008425063,-0.624468425604734,-0.24158180554755,0.267985636792218],[0,0,0,0],[8.999999E+09,8.999999E+09,8.999999E+09,8.999999E+09,8.999999E+09,8.999999E+09]];
	LOCAL CONST Robtarget Tr_meulage_bavure_P149 :=[[117.834921875,-97.4784140625,99.0858671875],[0.693860106096755,-0.625065696308637,-0.239321899891789,0.265661545387704],[0,0,0,0],[8.999999E+09,8.999999E+09,8.999999E+09,8.999999E+09,8.999999E+09,8.999999E+09]];
	LOCAL CONST Robtarget Tr_meulage_bavure_P150 :=[[118.20546875,-97.0861484375,98.995765625],[0.69453428431535,-0.625551456780357,-0.2378473467914,0.264076016432445],[0,0,0,0],[8.999999E+09,8.999999E+09,8.999999E+09,8.999999E+09,8.999999E+09,8.999999E+09]];
	LOCAL CONST Robtarget Tr_meulage_bavure_P151 :=[[118.7105390625,-96.6043671875,98.8796796875],[0.694620371104656,-0.625831818173955,-0.237446491102241,0.263545516506628],[0,0,0,0],[8.999999E+09,8.999999E+09,8.999999E+09,8.999999E+09,8.999999E+09,8.999999E+09]];
	LOCAL CONST Robtarget Tr_meulage_bavure_P152 :=[[122.0213515625,-93.3379921875,98.1049453125],[0.694110464328635,-0.625900828376071,-0.23814331245253,0.264095776342168],[0,0,0,0],[8.999999E+09,8.999999E+09,8.999999E+09,8.999999E+09,8.999999E+09,8.999999E+09]];
	LOCAL CONST Robtarget Tr_meulage_bavure_P153 :=[[123.6533515625,-92.0036796875,97.75809375],[0.69309502723853,-0.62583427102132,-0.239723301434203,0.265487263690596],[0,0,0,0],[8.999999E+09,8.999999E+09,8.999999E+09,8.999999E+09,8.999999E+09,8.999999E+09]];
	LOCAL CONST Robtarget Tr_meulage_bavure_P154 :=[[126.4854140625,-89.31546875,97.1088359375],[0.691725305191532,-0.625743111934647,-0.241843548861069,0.267345016595241],[0,0,0,0],[8.999999E+09,8.999999E+09,8.999999E+09,8.999999E+09,8.999999E+09,8.999999E+09]];
	LOCAL CONST Robtarget Tr_meulage_bavure_P155 :=[[126.716828125,-89.086875,97.0546484375],[0.690157272035873,-0.625734721317842,-0.244163461223947,0.269301323049901],[0,0,0,0],[8.999999E+09,8.999999E+09,8.999999E+09,8.999999E+09,8.999999E+09,8.999999E+09]];
	LOCAL CONST Robtarget Tr_meulage_bavure_P156 :=[[126.9091640625,-88.89065625,97.0088203125],[0.688519981337476,-0.625884701298253,-0.246421065114997,0.271081601455039],[0,0,0,0],[8.999999E+09,8.999999E+09,8.999999E+09,8.999999E+09,8.999999E+09,8.999999E+09]];
	LOCAL CONST Robtarget Tr_meulage_bavure_P157 :=[[130.2696875,-85.3358828125,96.1920390625],[0.686899161746463,-0.626225517621117,-0.248464264125009,0.272537432520724],[0,0,0,0],[8.999999E+09,8.999999E+09,8.999999E+09,8.999999E+09,8.999999E+09,8.999999E+09]];
	LOCAL CONST Robtarget Tr_meulage_bavure_P158 :=[[134.441171875,-81.065984375,95.19628125],[0.685336873912411,-0.626755183413547,-0.250238321528855,0.27362765167036],[0,0,0,0],[8.999999E+09,8.999999E+09,8.999999E+09,8.999999E+09,8.999999E+09,8.999999E+09]];
	LOCAL CONST Robtarget Tr_meulage_bavure_P159 :=[[135.270625,-80.214390625,94.9979609375],[0.683854866948306,-0.627434135833296,-0.251751844694846,0.274390114317157],[0,0,0,0],[8.999999E+09,8.999999E+09,8.999999E+09,8.999999E+09,8.999999E+09,8.999999E+09]];
	LOCAL CONST Robtarget Tr_meulage_bavure_P160 :=[[135.577703125,-79.9067890625,94.925515625],[0.682441617542514,-0.628212789839451,-0.25306919678964,0.27491473398917],[0,0,0,0],[8.999999E+09,8.999999E+09,8.999999E+09,8.999999E+09,8.999999E+09,8.999999E+09]];
	LOCAL CONST Robtarget Tr_meulage_bavure_P161 :=[[137.737515625,-77.7647109375,94.4186875],[0.681081783472603,-0.629037728160835,-0.254262586378242,0.27529925161591],[0,0,0,0],[8.999999E+09,8.999999E+09,8.999999E+09,8.999999E+09,8.999999E+09,8.999999E+09]];
	LOCAL CONST Robtarget Tr_meulage_bavure_P162 :=[[138.148109375,-77.372625,94.3242578125],[0.679775149432518,-0.629852651567216,-0.255384692418076,0.275626635879533],[0,0,0,0],[8.999999E+09,8.999999E+09,8.999999E+09,8.999999E+09,8.999999E+09,8.999999E+09]];
	LOCAL CONST Robtarget Tr_meulage_bavure_P163 :=[[139.75109375,-75.7219375,93.940359375],[0.678526211998911,-0.630631190802711,-0.256453866383674,0.275930960992107],[0,0,0,0],[8.999999E+09,8.999999E+09,8.999999E+09,8.999999E+09,8.999999E+09,8.999999E+09]];
	LOCAL CONST Robtarget Tr_meulage_bavure_P164 :=[[144.222375,-71.20096875,92.8801328125],[0.677351276572553,-0.63136681903535,-0.25745338234804,0.276204532664239],[0,0,0,0],[8.999999E+09,8.999999E+09,8.999999E+09,8.999999E+09,8.999999E+09,8.999999E+09]];
	LOCAL CONST Robtarget Tr_meulage_bavure_P165 :=[[146.255125,-69.1668515625,92.4008203125],[0.67627107054316,-0.632066051641482,-0.258348321411361,0.276416516027331],[0,0,0,0],[8.999999E+09,8.999999E+09,8.999999E+09,8.999999E+09,8.999999E+09,8.999999E+09]];
	LOCAL CONST Robtarget Tr_meulage_bavure_P166 :=[[147.403828125,-68.0020078125,92.128015625],[0.67530954855657,-0.632727226620558,-0.259106820005068,0.276544618729491],[0,0,0,0],[8.999999E+09,8.999999E+09,8.999999E+09,8.999999E+09,8.999999E+09,8.999999E+09]];
	LOCAL CONST Robtarget Tr_meulage_bavure_P167 :=[[149.368375,-65.896875,91.64709375],[0.674474542514208,-0.633344388379192,-0.259723959168028,0.276590748657511],[0,0,0,0],[8.999999E+09,8.999999E+09,8.999999E+09,8.999999E+09,8.999999E+09,8.999999E+09]];
	LOCAL CONST Robtarget Tr_meulage_bavure_P168 :=[[151.09534375,-64.10015234375,91.2311640625],[0.673758315919046,-0.633913814116057,-0.26021480240699,0.276570541835271],[0,0,0,0],[8.999999E+09,8.999999E+09,8.999999E+09,8.999999E+09,8.999999E+09,8.999999E+09]];
	LOCAL CONST Robtarget Tr_meulage_bavure_P169 :=[[151.4521875,-63.70352734375,91.142],[0.673151768417488,-0.634426133549226,-0.260601465313278,0.276508687065633],[0,0,0,0],[8.999999E+09,8.999999E+09,8.999999E+09,8.999999E+09,8.999999E+09,8.999999E+09]];
	LOCAL CONST Robtarget Tr_meulage_bavure_P170 :=[[158.654796875,-56.5154296875,89.446140625],[0.672649092526845,-0.634885417789131,-0.260888842912173,0.27640679486127],[0,0,0,0],[8.999999E+09,8.999999E+09,8.999999E+09,8.999999E+09,8.999999E+09,8.999999E+09]];
	LOCAL CONST Robtarget Tr_meulage_bavure_P171 :=[[160.33015625,-54.912390625,89.0604296875],[0.67227088900005,-0.635301400744327,-0.261038950014287,0.276229340568334],[0,0,0,0],[8.999999E+09,8.999999E+09,8.999999E+09,8.999999E+09,8.999999E+09,8.999999E+09]];
	LOCAL CONST Robtarget Tr_meulage_bavure_P172 :=[[161.691203125,-53.386296875,88.7186484375],[0.6720457760073,-0.635704408750129,-0.260982989347098,0.275902625790056],[0,0,0,0],[8.999999E+09,8.999999E+09,8.999999E+09,8.999999E+09,8.999999E+09,8.999999E+09]];
	LOCAL CONST Robtarget Tr_meulage_bavure_P173 :=[[166.187515625,-48.72094921875,87.637359375],[0.672001971888506,-0.636134297133524,-0.260643129242391,0.275339181678037],[0,0,0,0],[8.999999E+09,8.999999E+09,8.999999E+09,8.999999E+09,8.999999E+09,8.999999E+09]];
	LOCAL CONST Robtarget Tr_meulage_bavure_P174 :=[[166.338609375,-48.56569140625,87.6012109375],[0.672167471379119,-0.636608577616384,-0.259961500401227,0.274482108040194],[0,0,0,0],[8.999999E+09,8.999999E+09,8.999999E+09,8.999999E+09,8.999999E+09,8.999999E+09]];
	LOCAL CONST Robtarget Tr_meulage_bavure_P175 :=[[166.41075,-48.4941171875,87.58428125],[0.672534798008807,-0.637132381341716,-0.258941022630752,0.273329143912662],[0,0,0,0],[8.999999E+09,8.999999E+09,8.999999E+09,8.999999E+09,8.999999E+09,8.999999E+09]];
	LOCAL CONST Robtarget Tr_meulage_bavure_P176 :=[[169.64184375,-45.33905078125,86.8323515625],[0.673073404765533,-0.637677124608727,-0.257648935193759,0.271950552015621],[0,0,0,0],[8.999999E+09,8.999999E+09,8.999999E+09,8.999999E+09,8.999999E+09,8.999999E+09]];
	LOCAL CONST Robtarget Tr_meulage_bavure_P177 :=[[171.828578125,-43.01941015625,86.30003125],[0.673733049918126,-0.638184254650028,-0.256210678504562,0.270482389047865],[0,0,0,0],[8.999999E+09,8.999999E+09,8.999999E+09,8.999999E+09,8.999999E+09,8.999999E+09]];
	LOCAL CONST Robtarget Tr_meulage_bavure_P178 :=[[172.766703125,-42.08340234375,86.0791796875],[0.674437765232538,-0.638588311058595,-0.254798705828694,0.269102748621215],[0,0,0,0],[8.999999E+09,8.999999E+09,8.999999E+09,8.999999E+09,8.999999E+09,8.999999E+09]];
	LOCAL CONST Robtarget Tr_meulage_bavure_P179 :=[[175.191515625,-39.7303359375,85.51675],[0.675114027600113,-0.638812936640071,-0.253596466276914,0.268007302159297],[0,0,0,0],[8.999999E+09,8.999999E+09,8.999999E+09,8.999999E+09,8.999999E+09,8.999999E+09]];
	LOCAL CONST Robtarget Tr_meulage_bavure_P180 :=[[178.975015625,-36.1385234375,84.6493125],[0.675692385374946,-0.63879602181101,-0.252770149648418,0.267369957757896],[0,0,0,0],[8.999999E+09,8.999999E+09,8.999999E+09,8.999999E+09,8.999999E+09,8.999999E+09]];
	LOCAL CONST Robtarget Tr_meulage_bavure_P181 :=[[180.91965625,-34.30773828125,84.2054140625],[0.676139585740671,-0.638491716843228,-0.252416732479546,0.267300170746991],[0,0,0,0],[8.999999E+09,8.999999E+09,8.999999E+09,8.999999E+09,8.999999E+09,8.999999E+09]];
	LOCAL CONST Robtarget Tr_meulage_bavure_P182 :=[[183.21415625,-32.2158125,83.6903203125],[0.676464091677058,-0.637893245736709,-0.252530539929744,0.267800048763646],[0,0,0,0],[8.999999E+09,8.999999E+09,8.999999E+09,8.999999E+09,8.999999E+09,8.999999E+09]];
	LOCAL CONST Robtarget Tr_meulage_bavure_P183 :=[[186.697203125,-28.652521484375,82.859140625],[0.676713579249591,-0.637037326727618,-0.253002416235379,0.268760029383087],[0,0,0,0],[8.999999E+09,8.999999E+09,8.999999E+09,8.999999E+09,8.999999E+09,8.999999E+09]];
	LOCAL CONST Robtarget Tr_meulage_bavure_P184 :=[[188.72565625,-26.596564453125,82.37753125],[0.676967536434926,-0.635989246301468,-0.253648101270113,0.269991247865898],[0,0,0,0],[8.999999E+09,8.999999E+09,8.999999E+09,8.999999E+09,8.999999E+09,8.999999E+09]];
	LOCAL CONST Robtarget Tr_meulage_bavure_P185 :=[[194.09678125,-21.243751953125,81.11384375],[0.677313909517489,-0.634811556993404,-0.254275933509896,0.271300395722925],[0,0,0,0],[8.999999E+09,8.999999E+09,8.999999E+09,8.999999E+09,8.999999E+09,8.999999E+09]];
	LOCAL CONST Robtarget Tr_meulage_bavure_P186 :=[[198.388484375,-16.9421875,80.101],[0.677791093328982,-0.633525087702924,-0.254808670809252,0.272612799287428],[0,0,0,0],[8.999999E+09,8.999999E+09,8.999999E+09,8.999999E+09,8.999999E+09,8.999999E+09]];
	LOCAL CONST Robtarget Tr_meulage_bavure_P187 :=[[201.41609375,-13.90492578125,79.3861484375],[0.678358513290387,-0.63207509649309,-0.255354487465879,0.27405270582635],[0,0,0,0],[8.999999E+09,8.999999E+09,8.999999E+09,8.999999E+09,8.999999E+09,8.999999E+09]];
	LOCAL CONST Robtarget Tr_meulage_bavure_P188 :=[[205.76146875,-9.5805009765625,78.3645703125],[0.678864723184876,-0.630308959727673,-0.256266855002795,0.276008336702204],[0,0,0,0],[8.999999E+09,8.999999E+09,8.999999E+09,8.999999E+09,8.999999E+09,8.999999E+09]];
	LOCAL CONST Robtarget Tr_meulage_bavure_P189 :=[[209.072,-6.3418076171875,77.5933828125],[0.679038620164077,-0.627961714197701,-0.258155355067428,0.279153095052806],[0,0,0,0],[8.999999E+09,8.999999E+09,8.999999E+09,8.999999E+09,8.999999E+09,8.999999E+09]];
	LOCAL CONST Robtarget Tr_meulage_bavure_P190 :=[[209.864234375,-5.56084423828125,77.408078125],[0.678461315398997,-0.624648328129081,-0.261894912721953,0.284456963990983],[0,0,0,0],[8.999999E+09,8.999999E+09,8.999999E+09,8.999999E+09,8.999999E+09,8.999999E+09]];
	LOCAL CONST Robtarget Tr_meulage_bavure_P191 :=[[210.8583125,-4.59485791015625,77.1773359375],[0.676601352748294,-0.619891149224572,-0.268472051853997,0.293032984398552],[0,0,0,0],[8.999999E+09,8.999999E+09,8.999999E+09,8.999999E+09,8.999999E+09,8.999999E+09]];
	LOCAL CONST Robtarget Tr_meulage_bavure_P192 :=[[212.803,-2.75844091796875,76.73271875],[0.672791648081798,-0.61311271595714,-0.278895068415668,0.30604205040559],[0,0,0,0],[8.999999E+09,8.999999E+09,8.999999E+09,8.999999E+09,8.999999E+09,8.999999E+09]];
	LOCAL CONST Robtarget Tr_meulage_bavure_P193 :=[[215.38290625,-0.307765075683594,76.1410390625],[0.666181213763021,-0.603587048693227,-0.294119766721531,0.324621052771845],[0,0,0,0],[8.999999E+09,8.999999E+09,8.999999E+09,8.999999E+09,8.999999E+09,8.999999E+09]];
	LOCAL CONST Robtarget Tr_meulage_bavure_P194 :=[[217.938078125,2.29241845703125,75.533046875],[0.655694163717862,-0.590404851222067,-0.314913624092562,0.349738022926692],[0,0,0,0],[8.999999E+09,8.999999E+09,8.999999E+09,8.999999E+09,8.999999E+09,8.999999E+09]];
	LOCAL CONST Robtarget Tr_meulage_bavure_P195 :=[[217.966234375,2.33756127929687,75.52425],[0.640014311942631,-0.572495200846076,-0.341666440245698,0.381961999584573],[0,0,0,0],[8.999999E+09,8.999999E+09,8.999999E+09,8.999999E+09,8.999999E+09,8.999999E+09]];
	LOCAL CONST Robtarget Tr_meulage_bavure_P196 :=[[219.655078125,4.75369140625,75.0337578125],[0.617802002978358,-0.548801016034438,-0.374000950268676,0.421024250030357],[0,0,0,0],[8.999999E+09,8.999999E+09,8.999999E+09,8.999999E+09,8.999999E+09,8.999999E+09]];
	LOCAL CONST Robtarget Tr_meulage_bavure_P197 :=[[219.958140625,5.72391552734375,74.877546875],[0.588173901173118,-0.518717257809693,-0.410401282914292,0.465354333182244],[0,0,0,0],[8.999999E+09,8.999999E+09,8.999999E+09,8.999999E+09,8.999999E+09,8.999999E+09]];
	LOCAL CONST Robtarget Tr_meulage_bavure_P198 :=[[220.410296875,7.4067080078125,74.6145859375],[0.551489052581509,-0.482748410649071,-0.448086207645967,0.511891148014889],[0,0,0,0],[8.999999E+09,8.999999E+09,8.999999E+09,8.999999E+09,8.999999E+09,8.999999E+09]];
	LOCAL CONST Robtarget Tr_meulage_bavure_P199 :=[[219.6829375,10.276052734375,74.3289921875],[0.509749535585182,-0.442815093807732,-0.483727635142197,0.556846279206818],[0,0,0,0],[8.999999E+09,8.999999E+09,8.999999E+09,8.999999E+09,8.999999E+09,8.999999E+09]];
	LOCAL CONST Robtarget Tr_meulage_bavure_P200 :=[[219.558859375,10.7425,74.2831953125],[0.466182432063737,-0.401845222204687,-0.514593552424609,0.59698227212324],[0,0,0,0],[8.999999E+09,8.999999E+09,8.999999E+09,8.999999E+09,8.999999E+09,8.999999E+09]];
	LOCAL CONST Robtarget Tr_meulage_bavure_P201 :=[[218.754390625,11.7430322265625,74.243453125],[0.424240719385272,-0.362857065115585,-0.53927625033867,0.630504312540236],[0,0,0,0],[8.999999E+09,8.999999E+09,8.999999E+09,8.999999E+09,8.999999E+09,8.999999E+09]];
	LOCAL CONST Robtarget Tr_meulage_bavure_P202 :=[[217.384296875,13.574150390625,74.159609375],[0.38686782802582,-0.328337560107026,-0.557585760739142,0.656982381561715],[0,0,0,0],[8.999999E+09,8.999999E+09,8.999999E+09,8.999999E+09,8.999999E+09,8.999999E+09]];
	LOCAL CONST Robtarget Tr_meulage_bavure_P203 :=[[217.113796875,13.9777421875,74.137703125],[0.356085097619458,-0.299905091294226,-0.570121885035361,0.676920509124129],[0,0,0,0],[8.999999E+09,8.999999E+09,8.999999E+09,8.999999E+09,8.999999E+09,8.999999E+09]];
	LOCAL CONST Robtarget Tr_meulage_bavure_P204 :=[[216.528375,14.542376953125,74.1295546875],[0.332841753404339,-0.278228800245241,-0.577861882945526,0.691289191397833],[0,0,0,0],[8.999999E+09,8.999999E+09,8.999999E+09,8.999999E+09,8.999999E+09,8.999999E+09]];
	LOCAL CONST Robtarget Tr_meulage_bavure_P205 :=[[215.232296875,15.6981689453125,74.123484375],[0.316990619757028,-0.263048307231682,-0.581897967557801,0.70122556313978],[0,0,0,0],[8.999999E+09,8.999999E+09,8.999999E+09,8.999999E+09,8.999999E+09,8.999999E+09]];
	LOCAL CONST Robtarget Tr_meulage_bavure_P206 :=[[210.91459375,19.667748046875,74.088109375],[0.307517820368432,-0.253390036778211,-0.583252540710594,0.707843734995247],[0,0,0,0],[8.999999E+09,8.999999E+09,8.999999E+09,8.999999E+09,8.999999E+09,8.999999E+09]];
	LOCAL CONST Robtarget Tr_meulage_bavure_P207 :=[[208.90846875,21.6279375,74.0569609375],[0.302856735062657,-0.247866691694607,-0.58283551514248,0.712139497194305],[0,0,0,0],[8.999999E+09,8.999999E+09,8.999999E+09,8.999999E+09,8.999999E+09,8.999999E+09]];
	LOCAL CONST Robtarget Tr_meulage_bavure_P208 :=[[204.18896875,26.22773046875,73.98515625],[0.301336672752366,-0.2450481704566,-0.581389189438382,0.714936510617962],[0,0,0,0],[8.999999E+09,8.999999E+09,8.999999E+09,8.999999E+09,8.999999E+09,8.999999E+09]];
	LOCAL CONST Robtarget Tr_meulage_bavure_P209 :=[[200.303265625,29.980283203125,73.9304296875],[0.30158698926557,-0.2437790891667,-0.579440369029792,0.716844405941346],[0,0,0,0],[8.999999E+09,8.999999E+09,8.999999E+09,8.999999E+09,8.999999E+09,8.999999E+09]];
	LOCAL CONST Robtarget Tr_meulage_bavure_P210 :=[[194.683875,35.65457421875,73.81984375],[0.302650931193952,-0.243276560798919,-0.577346700693944,0.718254631736615],[0,0,0,0],[8.999999E+09,8.999999E+09,8.999999E+09,8.999999E+09,8.999999E+09,8.999999E+09]];
	LOCAL CONST Robtarget Tr_meulage_bavure_P211 :=[[190.825265625,39.4054921875,73.7623828125],[0.303954376487452,-0.243077209685885,-0.575315974430214,0.719400261822903],[0,0,0,0],[8.999999E+09,8.999999E+09,8.999999E+09,8.999999E+09,8.999999E+09,8.999999E+09]];
	LOCAL CONST Robtarget Tr_meulage_bavure_P212 :=[[182.394671875,47.662078125,73.6290546875],[0.305152524764486,-0.242912306473418,-0.573477072615034,0.720416265209577],[0,0,0,0],[8.999999E+09,8.999999E+09,8.999999E+09,8.999999E+09,8.999999E+09,8.999999E+09]];
	LOCAL CONST Robtarget Tr_meulage_bavure_P213 :=[[182.047609375,48.00865625,73.62271875],[0.306062082928783,-0.242646131684416,-0.571903015991084,0.721370776003704],[0,0,0,0],[8.999999E+09,8.999999E+09,8.999999E+09,8.999999E+09,8.999999E+09,8.999999E+09]];
	LOCAL CONST Robtarget Tr_meulage_bavure_P214 :=[[181.94528125,48.11698828125,73.6200625],[0.306538641667199,-0.242170039014412,-0.57064599935653,0.722323249512968],[0,0,0,0],[8.999999E+09,8.999999E+09,8.999999E+09,8.999999E+09,8.999999E+09,8.999999E+09]];
	LOCAL CONST Robtarget Tr_meulage_bavure_P215 :=[[174.51259375,55.72409765625,73.460859375],[0.306478671066334,-0.241408566105795,-0.569744077747358,0.72331487905612],[0,0,0,0],[8.999999E+09,8.999999E+09,8.999999E+09,8.999999E+09,8.999999E+09,8.999999E+09]];
	LOCAL CONST Robtarget Tr_meulage_bavure_P216 :=[[170.818171875,59.35505859375,73.4008046875],[0.30587018954178,-0.240354753367828,-0.569199788732217,0.724351171870637],[0,0,0,0],[8.999999E+09,8.999999E+09,8.999999E+09,8.999999E+09,8.999999E+09,8.999999E+09]];
	LOCAL CONST Robtarget Tr_meulage_bavure_P217 :=[[167.61278125,62.55397265625,73.34253125],[0.304804023906887,-0.23907661194975,-0.568975341300375,0.725399160201417],[0,0,0,0],[8.999999E+09,8.999999E+09,8.999999E+09,8.999999E+09,8.999999E+09,8.999999E+09]];
	LOCAL CONST Robtarget Tr_meulage_bavure_P218 :=[[166.61040625,63.48946484375,73.332546875],[0.303467389409373,-0.237718453627246,-0.569004878835783,0.726382081435938],[0,0,0,0],[8.999999E+09,8.999999E+09,8.999999E+09,8.999999E+09,8.999999E+09,8.999999E+09]];
	LOCAL CONST Robtarget Tr_meulage_bavure_P219 :=[[164.6754375,65.5178125,73.285],[0.30212332843895,-0.236470421121618,-0.569183249181315,0.727209504337599],[0,0,0,0],[8.999999E+09,8.999999E+09,8.999999E+09,8.999999E+09,8.999999E+09,8.999999E+09]];
	LOCAL CONST Robtarget Tr_meulage_bavure_P220 :=[[164.027875,66.1586171875,73.273921875],[0.30100699155398,-0.235501992323817,-0.569418376113346,0.727802387734181],[0,0,0,0],[8.999999E+09,8.999999E+09,8.999999E+09,8.999999E+09,8.999999E+09,8.999999E+09]];
	LOCAL CONST Robtarget Tr_meulage_bavure_P221 :=[[162.604015625,67.4741875,73.2614296875],[0.300151428597899,-0.234819642455501,-0.569677264391283,0.728173516315566],[0,0,0,0],[8.999999E+09,8.999999E+09,8.999999E+09,8.999999E+09,8.999999E+09,8.999999E+09]];
	LOCAL CONST Robtarget Tr_meulage_bavure_P222 :=[[158.595015625,71.3477890625,73.20471875],[0.299321838371479,-0.234219549306674,-0.570010582536318,0.728447373248819],[0,0,0,0],[8.999999E+09,8.999999E+09,8.999999E+09,8.999999E+09,8.999999E+09,8.999999E+09]];
	LOCAL CONST Robtarget Tr_meulage_bavure_P223 :=[[157.051328125,72.876828125,73.1781171875],[0.297950406092332,-0.233235099365498,-0.570571161863959,0.728886474824847],[0,0,0,0],[8.999999E+09,8.999999E+09,8.999999E+09,8.999999E+09,8.999999E+09,8.999999E+09]];
	LOCAL CONST Robtarget Tr_meulage_bavure_P224 :=[[156.589515625,73.2621328125,73.1793203125],[0.295196830881914,-0.231188115066846,-0.571597187514496,0.729854466119535],[0,0,0,0],[8.999999E+09,8.999999E+09,8.999999E+09,8.999999E+09,8.999999E+09,8.999999E+09]];
	LOCAL CONST Robtarget Tr_meulage_bavure_P225 :=[[155.77396875,73.908546875,73.18578125],[0.290165323897004,-0.227351684500612,-0.573322171425624,0.731721930868747],[0,0,0,0],[8.999999E+09,8.999999E+09,8.999999E+09,8.999999E+09,8.999999E+09,8.999999E+09]];
	LOCAL CONST Robtarget Tr_meulage_bavure_P226 :=[[153.8596875,75.6487734375,73.1726015625],[0.282116404029001,-0.221124035757434,-0.575898824815611,0.73474828272279],[0,0,0,0],[8.999999E+09,8.999999E+09,8.999999E+09,8.999999E+09,8.999999E+09,8.999999E+09]];
	LOCAL CONST Robtarget Tr_meulage_bavure_P227 :=[[149.35040625,80.1121171875,73.095296875],[0.270786830527884,-0.21228353590668,-0.579291902061702,0.73893916190804],[0,0,0,0],[8.999999E+09,8.999999E+09,8.999999E+09,8.999999E+09,8.999999E+09,8.999999E+09]];
	LOCAL CONST Robtarget Tr_meulage_bavure_P228 :=[[140.9526875,88.5314609375,72.9377109375],[0.25653662041413,-0.201112154641619,-0.583264519500213,0.744006292939843],[0,0,0,0],[8.999999E+09,8.999999E+09,8.999999E+09,8.999999E+09,8.999999E+09,8.999999E+09]];
	LOCAL CONST Robtarget Tr_meulage_bavure_P229 :=[[139.3685625,90.184125,72.899796875],[0.2403454168092,-0.188377955306203,-0.587413412962929,0.749462012943091],[0,0,0,0],[8.999999E+09,8.999999E+09,8.999999E+09,8.999999E+09,8.999999E+09,8.999999E+09]];
	LOCAL CONST Robtarget Tr_meulage_bavure_P230 :=[[138.703984375,90.7161875,72.9043828125],[0.223667222335745,-0.175228811204284,-0.591293703340151,0.754744720926775],[0,0,0,0],[8.999999E+09,8.999999E+09,8.999999E+09,8.999999E+09,8.999999E+09,8.999999E+09]];
	LOCAL CONST Robtarget Tr_meulage_bavure_P231 :=[[137.47715625,91.81784375,72.8976640625],[0.208103420685467,-0.162932534107107,-0.594548907411586,0.759379715507422],[0,0,0,0],[8.999999E+09,8.999999E+09,8.999999E+09,8.999999E+09,8.999999E+09,8.999999E+09]];
	LOCAL CONST Robtarget Tr_meulage_bavure_P232 :=[[135.177359375,93.092203125,72.9855703125],[0.195192880749293,-0.152709960778427,-0.596960883410108,0.763031526781212],[0,0,0,0],[8.999999E+09,8.999999E+09,8.999999E+09,8.999999E+09,8.999999E+09,8.999999E+09]];
	LOCAL CONST Robtarget Tr_meulage_bavure_P233 :=[[134.71934375,93.369140625,73.0001328125],[0.186305547507915,-0.145644225992654,-0.598419687251703,0.765488001416319],[0,0,0,0],[8.999999E+09,8.999999E+09,8.999999E+09,8.999999E+09,8.999999E+09,8.999999E+09]];
	LOCAL CONST Robtarget Tr_meulage_bavure_P234 :=[[132.566421875,94.0453203125,73.14809375],[0.182530709465366,-0.142594677973167,-0.598882115772344,0.76660909812227],[0,0,0,0],[8.999999E+09,8.999999E+09,8.999999E+09,8.999999E+09,8.999999E+09,8.999999E+09]];
	LOCAL CONST Robtarget Tr_meulage_bavure_P235 :=[[130.75496875,94.7049609375,73.2610546875],[0.184484856712306,-0.144051668822647,-0.598343359223879,0.76628955286232],[0,0,0,0],[8.999999E+09,8.999999E+09,8.999999E+09,8.999999E+09,8.999999E+09,8.999999E+09]];
	LOCAL CONST Robtarget Tr_meulage_bavure_P236 :=[[126.546109375,96.0332421875,73.5495],[0.192057864060522,-0.149943635957893,-0.596838158277242,0.76447033671194],[0,0,0,0],[8.999999E+09,8.999999E+09,8.999999E+09,8.999999E+09,8.999999E+09,8.999999E+09]];
	LOCAL CONST Robtarget Tr_meulage_bavure_P237 :=[[124.82028125,96.897859375,73.627109375],[0.20433127139178,-0.159580623171283,-0.594470161855184,0.761175395624133],[0,0,0,0],[8.999999E+09,8.999999E+09,8.999999E+09,8.999999E+09,8.999999E+09,8.999999E+09]];
	LOCAL CONST Robtarget Tr_meulage_bavure_P238 :=[[123.6533359375,97.510421875,73.676046875],[0.219594421243523,-0.171665070482128,-0.591474460610111,0.756615725570825],[0,0,0,0],[8.999999E+09,8.999999E+09,8.999999E+09,8.999999E+09,8.999999E+09,8.999999E+09]];
	LOCAL CONST Robtarget Tr_meulage_bavure_P239 :=[[122.768828125,98.07971875,73.6997890625],[0.235670229676833,-0.184546283771791,-0.588265409617017,0.751229671830269],[0,0,0,0],[8.999999E+09,8.999999E+09,8.999999E+09,8.999999E+09,8.999999E+09,8.999999E+09]];
	LOCAL CONST Robtarget Tr_meulage_bavure_P240 :=[[120.9908671875,99.4119921875,73.723640625],[0.250251631871621,-0.19646022024423,-0.585412779780119,0.745700596672213],[0,0,0,0],[8.999999E+09,8.999999E+09,8.999999E+09,8.999999E+09,8.999999E+09,8.999999E+09]];
	LOCAL CONST Robtarget Tr_meulage_bavure_P241 :=[[120.4433359375,99.899390625,73.7211875],[0.26093230713188,-0.205542482161428,-0.583662487414019,0.740948527164629],[0,0,0,0],[8.999999E+09,8.999999E+09,8.999999E+09,8.999999E+09,8.999999E+09,8.999999E+09]];
	LOCAL CONST Robtarget Tr_meulage_bavure_P242 :=[[112.005375,108.5710390625,73.5359140625],[0.265347774125823,-0.209924489100336,-0.583851417783083,0.737997147416654],[0,0,0,0],[8.999999E+09,8.999999E+09,8.999999E+09,8.999999E+09,8.999999E+09,8.999999E+09]];
	LOCAL CONST Robtarget Tr_meulage_bavure_P243 :=[[111.7476484375,108.8401171875,73.52971875],[0.261165617566264,-0.207694077912816,-0.586755085977258,0.737817158434932],[0,0,0,0],[8.999999E+09,8.999999E+09,8.999999E+09,8.999999E+09,8.999999E+09,8.999999E+09]];
	LOCAL CONST Robtarget Tr_meulage_bavure_P244 :=[[111.5534140625,109.058109375,73.5231171875],[0.246136019502772,-0.196925309056293,-0.592877885437413,0.741035286282425],[0,0,0,0],[8.999999E+09,8.999999E+09,8.999999E+09,8.999999E+09,8.999999E+09,8.999999E+09]];
	LOCAL CONST Robtarget Tr_meulage_bavure_P245 :=[[107.021359375,114.0215234375,73.3847421875],[0.218342524018878,-0.175872067380629,-0.602138479675959,0.747545857733058],[0,0,0,0],[8.999999E+09,8.999999E+09,8.999999E+09,8.999999E+09,8.999999E+09,8.999999E+09]];
	LOCAL CONST Robtarget Tr_meulage_bavure_P246 :=[[105.0492109375,115.6444296875,73.392765625],[0.176696299249378,-0.143369462155227,-0.613544655952204,0.756165702941747],[0,0,0,0],[8.999999E+09,8.999999E+09,8.999999E+09,8.999999E+09,8.999999E+09,8.999999E+09]];
	LOCAL CONST Robtarget Tr_meulage_bavure_P247 :=[[104.4821328125,116.109125,73.3953125],[0.121984655509143,-0.0997398047164254,-0.625080142053884,0.764491027537499],[0,0,0,0],[8.999999E+09,8.999999E+09,8.999999E+09,8.999999E+09,8.999999E+09,8.999999E+09]];
	LOCAL CONST Robtarget Tr_meulage_bavure_P248 :=[[102.1142421875,117.360921875,73.493484375],[0.0579279405228145,-0.047737024426932,-0.634164384459843,0.769546011417327],[0,0,0,0],[8.999999E+09,8.999999E+09,8.999999E+09,8.999999E+09,8.999999E+09,8.999999E+09]];
	LOCAL CONST Robtarget Tr_meulage_bavure_P249 :=[[101.4949609375,117.718609375,73.5153046875],[0.00904115723472132,-0.00750847395762135,0.638842591669632,-0.769247699615353],[0,0,0,0],[8.999999E+09,8.999999E+09,8.999999E+09,8.999999E+09,8.999999E+09,8.999999E+09]];
	LOCAL CONST Robtarget Tr_meulage_bavure_P250 :=[[98.2574921875,117.9863515625,73.832984375],[0.0721652468811392,-0.0603755494160705,0.638828320563473,-0.763574061254928],[0,0,0,0],[8.999999E+09,8.999999E+09,8.999999E+09,8.999999E+09,8.999999E+09,8.999999E+09]];
